ELSIF G_xDoManual THEN
	IF G_xManualActive AND G_xManualEpas AND IFB_RTOPMode.Q THEN
		G_xManualActive := FALSE;
		G_xManualEpas := FALSE;
	ELSIF IFB_RTOPMode.Q THEN
		g_xManualActive := TRUE;
		G_xManualEpas := TRUE;
	END_IF
	G_xJogMachineEpas := FALSE;
	G_xBrakeReleaseEpas := FALSE;
	G_xPrepareEpas:= FALSE;
	G_xAutoEpas := FALSE;

ELSIF g_xDoJogMachine THEN
	IF g_xJogMachineActive AND G_xJogMachineEpas AND IFB_RTOPMode.Q THEN
		g_xJogMachineActive := FALSE;
		G_xJogMachineEpas := FALSE;
	ELSIF IFB_RTOPMode.Q THEN
		g_xJogMachineActive := TRUE;
		G_xJogMachineEpas := TRUE;
	END_IF
	G_xBrakeReleaseEpas := FALSE;
	G_xPrepareEpas:= FALSE;
	G_xAutoEpas := FALSE;
	G_xManualEpas := FALSE;

ELSIF g_xDoBrakeRelease THEN
	IF g_xBrakeReleaseActive AND G_xBrakeReleaseEpas AND IFB_RTOPMode.Q THEN
		g_xBrakeReleaseActive := FALSE;
		G_xBrakeReleaseEpas := FALSE;
	ELSIF IFB_RTOPMode.Q THEN
		g_xBrakeReleaseActive := TRUE;
		G_xBrakeReleaseEpas := TRUE;
	END_IF
	G_xPrepareEpas:= FALSE;
	G_xAutoEpas := FALSE;
	G_xManualEpas := FALSE;
	G_xJogMachineEpas := FALSE;
END_IF

IF g_xDoPrepare OR  g_xDoAuto OR g_xDoManual OR g_xDoJogMachine OR g_xDoBrakeRelease THEN
	g_xPrepareActive := g_xPrepareActive  AND NOT( g_xDoAuto OR g_xDoManual OR g_xDoJogMachine OR g_xDoBrakeRelease);
	g_xAutoActive :=  g_xAutoActive AND NOT( g_xDoPrepare OR g_xDoManual OR g_xDoJogMachine OR g_xDoBrakeRelease);
	g_xManualActive := g_xManualActive AND NOT( g_xDoPrepare OR g_xDoAuto OR g_xDoJogMachine OR g_xDoBrakeRelease);
	g_xJogMachineActive :=  g_xJogMachineActive AND NOT( g_xDoPrepare OR g_xDoAuto OR g_xDoManual OR g_xDoBrakeRelease);
	g_xBrakeReleaseActive:=  g_xBrakeReleaseActive  AND NOT( g_xDoPrepare OR g_xDoAuto OR g_xDoManual OR g_xDoJogMachine);
END_IF
END_ACTION

ACTION SearchCurrentModule:
(* Locate the current module according to the information in audiHierarchy *)
udiCurrentLevel3Size := 0;
pstCurrentFirstLevel3Module := 0;
pstCurrentParent := 0;
dwCurrentAddInterface := 0;
pstCurrent := ADR(SR_MainMachine.stMachineInterface); (* here we have to start at SR_MainMachine.stMachineInterface
instead of our local copy because otherwise it would not be possible to send commands to the MainMachine using the Vis. *)
FOR udiTmp := 2 TO udiCurrentLevel DO
	(* Only navigate to existing modules *)
	IF(pstCurrent^.iq_stExt.udiNumberOfSubModules + pstCurrent^.iq_stExt.udiNumberOfControlModules < audiHierarchy[udiTmp]) THEN
		audiHierarchy[udiTmp] := pstCurrent^.iq_stExt.udiNumberOfSubModules + pstCurrent^.iq_stExt.udiNumberOfControlModules;
	END_IF
	IF(audiHierarchy[udiTmp] <= 0) THEN
		audiHierarchy[udiTmp] := 1;
	END_IF
	IF(pstCurrent^.iq_stExt.udiNumberOfSubModules = 0 AND pstCurrent^.iq_stExt.udiNumberOfControlModules = 0) THEN
		(* Stop, the hierarchy was invalid *)
		udiCurrentLevel := udiTmp - 1;
	ELSE
		(* In case the stSubModules structure of this module is invalid, create an error and stop *)
		IF(pstCurrent^.iq_stExt.dwSubModulesItf = 0) THEN
			stPointerException.sMsg:=						'SR_VisControl: dwSubModuleInterfaces of module was 0';
		END_IF
		IF (pstCurrent^.iq_stExt.pdwSubModulesAddItf = 0 AND pstCurrent^.iq_stExt.dwControlModulesItf = 0) THEN
			stPointerException.sMsg:=						'SR_VisControl: pdwSubModuleAddInterfaces of module was 0';
		END_IF
		(*Set an error if there is no sub module (control module or equipment module)*)
		IF( (pstCurrent^.iq_stExt.dwSubModulesItf = 0 )
			OR (pstCurrent^.iq_stExt.pdwSubModulesAddItf = 0) ) AND pstCurrent^.iq_stExt.dwControlModulesItf = 0 THEN
			(* Error, the structures are not set in the expected way *)
		
			stPointerException.etDiag			:= GD.ET_Diag.UnexpectedProgramBehavior;
			stPointerException.udiDiagExt		:= ET_DiagExt.InvalidPointer;
			stPointerException.sDiagExt			:= FC_EtDiagExtToString(stPointerException.udiDiagExt);
//			stPointerException.sMsg				:= '';
			stPointerException.udiModuleId		:= pstCurrent^.i_udiModuleId;
			stPointerException.sModuleName		:= pstCurrent^.i_sModuleName;
			stPointerException.etSource			:= TPL.ET_ExceptionSource.Vis;
			stPointerException.timDelayTime		:= T#0MS;
			stPointerException.wHmiAttributes	:= 0;
			stPointerException.xAutoQuit		:= FALSE;
			stPointerException.stReaction.axReaction[TPL.ET_Reaction.AsyncStop] := TRUE;

			TPL.FC_SetException(i_xExceptionActive	:= TRUE,
								iq_stException		:= stPointerException,
								iq_stExceptionList	:= G_stExceptionList,
								iq_stLogDataList	:= G_stLogDataList);
								
			xPointerExceptionActive := TRUE;
			RETURN;
		END_IF
		
		pstCurrentParent := pstCurrent;
		(* Only navigate to existing equipment modules *)
		IF pstCurrentParent^.iq_stExt.udiNumberOfSubModules >= audiHierarchy[udiTmp] THEN
			pstCurrent := pstCurrent^.iq_stExt.dwSubModulesItf
				+ UDINT_TO_DWORD((audiHierarchy[udiTmp] - 1) * SIZEOF(vpq_stCurrentModuleStandardInterface));
			IF(udiTmp = 2) THEN
				udiCurrentLevel3Size := pstCurrent^.iq_stExt.udiNumberOfSubModules;
				pstCurrentFirstLevel3Module := pstCurrent^.iq_stExt.dwSubModulesItf;
			END_IF
		END_IF
		(*Initialize pointer for level 2*)
		IF udiTmp = 2 THEN
			pstCurrentLevel2 := pstCurrent;
		END_IF

	END_IF
END_FOR

(*Set pointer to the current module interface*)
IF pstCurrentParent = 0  THEN
	pstCurrentControlModuleStandardInterface 	:= pstCurrent^.iq_stExt.dwControlModulesItf;
	udiCurrentNumberOfControlModules 			:= pstCurrent^.iq_stExt.udiNumberOfControlModules;
ELSE
	pstCurrentControlModuleStandardInterface 	:= pstCurrentParent^.iq_stExt.dwControlModulesItf;
	udiCurrentNumberOfControlModules 			:= pstCurrentParent^.iq_stExt.udiNumberOfControlModules;
END_IF
IF pstCurrentLevel2 <> 0 THEN
	udiNumberOfControlModulesLevel2:= pstCurrentLevel2^.iq_stExt.udiNumberOfControlModules;
ELSE
	udiNumberOfControlModulesLevel2:= 0;
END_IF
END_ACTION

ACTION SetCurrentModule:
(*
	handles all requests coming from the special vis controllers

	sets the current module by modifying aiHierachy
	also sets the jog target

inputs:
	diSetAsCurrentModule - if <> 0 contains the module ID of the module to set as current module

in_out:
	audiHierarchy	
	udiCurrentLevel

flags:
	

*)
IF(udiSetAsCurrentModule > 0) THEN
	udiTmp2 := 1;
	WHILE(udiSetAsCurrentModule > udiTmp2 * 100) DO
		udiTmp2 := udiTmp2 * 100;
	END_WHILE

	udiCurrentLevel := 0;
	WHILE(udiTmp2 > 0) DO
		udiCurrentLevel := udiCurrentLevel + 1;
		audiHierarchy[udiCurrentLevel] := udiSetAsCurrentModule / udiTmp2;
		udiSetAsCurrentModule := udiSetAsCurrentModule MOD udiTmp2;
		udiTmp2 := udiTmp2 / 100;
	END_WHILE

	IF(udiCurrentLevel < 1) THEN
		udiCurrentLevel := 1;
	END_IF

	udiSetAsCurrentModule := 0;
	xUpdateData := TRUE;
END_IF

IF(udiSetAsJogTarget <> 0) THEN
	G_udiManualModuleSelect		:= udiSetAsJogTarget;
//	G_udiManualElementSelect	:= udiSetAsJogTargetNum;
	udiSetAsJogTarget := 0;
//	udiSetAsJogTargetNum := 0;
END_IF
END_ACTION

END_PROGRAM

// LMC_PacDrive/Application/FB_ExampleLeafModuleVisController
FUNCTION_BLOCK FB_ExampleLeafModuleVisController

VAR_INPUT
	i_xEnable								: BOOL;
	i_pstMachineStandardItf					: POINTER TO TPL.ST_StandardModuleInterface;
	i_pstCurrentStandardItf					: POINTER TO TPL.ST_StandardModuleInterface;
	i_dwCurrentAddItf						: DWORD;
	i_xUpdateData							: BOOL; (* Signals the selection of another module *)
	i_udiCurrentJogTarget					: UDINT;
END_VAR

VAR_IN_OUT
	iq_stExceptionList				: TPL.ST_ExceptionList;
	iq_stLogDataList	   			: TPL.ST_LogDataList;
END_VAR

VAR_OUTPUT
	q_xActive								: BOOL;
	q_xReady								: BOOL;
	q_etDiag								: GD.ET_Diag := GD.ET_Diag.Ok;
	q_etDiagExt								: ET_DiagExtExampleLeafModule := ET_DiagExtExampleLeafModule.Disabled;
	q_sMsg									: STRING[80] := '';
	q_udiSetAsCurrentModule					: UDINT; (* A moduleID, if <> 0, it is set as the current module *)
	q_udiSetAsJogTarget						: UDINT;
END_VAR

VAR
	xCurrentIsOfMyType						: BOOL;
	pstCurrentExampleLeafModuleInterface	: POINTER TO ST_ExampleLeafModuleInterface;
	stCurrentExampleLeafModuleInterface		: ST_ExampleLeafModuleInterface;
	iPaneSelect								: INT := 1; (* Variable for selecting the active pane *)

	(* Variables to detect user changes in the vis *)
	xInitUserInputs							: BOOL;

	(* list of all example leaf modules in the machine *)
	audiExampleLeafModuleId					: ARRAY[1..c_udiMaxExampleLeafModules] OF UDINT; (* if <> 0, module exists *)
	asExampleLeafModuleName					: ARRAY[1..c_udiMaxExampleLeafModules] OF STRING[80]; (* if <> 0, module exists *)
	udiCountExampleLeafModules				: UDINT;
	udiSetAsCurrentModule					: UDINT;

	(* temporary variable, not to be used after init *)
	apExampleLeafModuleInterface			: ARRAY[1..c_udiMaxExampleLeafModules] OF POINTER TO TPL.ST_StandardModuleInterface;
	udiTmp									: UDINT;
	xEnableFlag								: BOOL;

	(* Variables to detect user changes in the vis *)
	lrPosMax								: LREAL;
END_VAR

VAR CONSTANT
	c_udiMaxExampleLeafModules : UDINT := 10;
END_VAR

q_udiSetAsCurrentModule 	:= 0;
q_udiSetAsJogTarget			:= 0;

(*********************************************************************)

IF i_xEnable AND NOT xEnableFlag THEN
	xEnableFlag := TRUE;
	
	q_xActive	:= TRUE;	
	
	q_etDiag	:= GD.ET_Diag.Ok;
	q_etDiagExt := ET_DiagExtExampleLeafModule.Initializing;
	q_sMsg		:= '';
	
	
		
	udiCountExampleLeafModules := TPL.FC_GetAllModulesOfType(	i_pstMachineStandardItf	:= i_pstMachineStandardItf,
																i_dwWantedType			:= ET_ModuleType.ExampleLeafModule,  
																i_pdwResultSet			:= ADR(apExampleLeafModuleInterface), 
																i_udiResultSetSize		:= c_udiMaxExampleLeafModules);
	FOR udiTmp := 1 TO udiCountExampleLeafModules DO
		(* module version check *)
		IF(apExampleLeafModuleInterface[udiTmp]^.q_udiModuleVersion = 1) THEN
			audiExampleLeafModuleId[udiTmp] := apExampleLeafModuleInterface[udiTmp]^.i_udiModuleId;
			asExampleLeafModuleName[udiTmp] := apExampleLeafModuleInterface[udiTmp]^.i_sModuleName;
		END_IF
	END_FOR
	
	q_xReady	:= TRUE;
	
	q_etDiag	:= GD.ET_Diag.Ok;
	q_etDiagExt	:= ET_DiagExtExampleLeafModule.Working;
	q_sMsg		:= '';
	
ELSIF NOT i_xEnable AND xEnableFlag THEN
	xEnableFlag := FALSE;
	
	q_xActive				:= FALSE;	
	q_xReady				:= FALSE;
	q_etDiag				:= GD.ET_Diag.Ok;
	q_etDiagExt				:= ET_DiagExtExampleLeafModule.Disabled;
	q_sMsg					:= '';
	q_udiSetAsCurrentModule	:= 0;		
	q_udiSetAsJogTarget		:= 0;		
END_IF

IF i_xEnable THEN
	q_udiSetAsCurrentModule := udiSetAsCurrentModule;
	udiSetAsCurrentModule := 0;
END_IF


(*********************************************************************)


IF i_xEnable THEN
	IF i_pstCurrentStandardItf = 0 THEN
		q_xReady := FALSE;
		q_etDiag := GD.ET_Diag.InputParameterInvalid;
		q_etDiagExt := ET_DiagExtExampleLeafModule.CurrentStandardItfInvalidPointer;
		q_sMsg := '';
	ELSIF i_dwCurrentAddItf = 0 THEN
		q_xReady := FALSE;
		q_etDiag := GD.ET_Diag.InputParameterInvalid;
		q_etDiagExt := ET_DiagExtExampleLeafModule.CurrentAddItfInvalidPointer;
		q_sMsg := '';
	ELSE
		q_xReady	:= TRUE;
	
		q_etDiag	:= GD.ET_Diag.Ok;
		q_etDiagExt	:= ET_DiagExtExampleLeafModule.Working;
		q_sMsg		:= '';
		
		IF (i_pstCurrentStandardItf^.q_dwModuleType = UDINT_TO_DWORD(ET_ModuleType.ExampleLeafModule)) THEN
			(* Module version check *)
			IF(i_pstCurrentStandardItf^.q_udiModuleVersion = 1) THEN
				pstCurrentExampleLeafModuleInterface := i_dwCurrentAddItf;
				xCurrentIsOfMyType := TRUE;
			END_IF
		ELSE
			pstCurrentExampleLeafModuleInterface := 0;
			xCurrentIsOfMyType := FALSE;
		END_IF	
	
		IF(xCurrentIsOfMyType) THEN
			(* Execute changes requested by user first *)
			IF(NOT xInitUserInputs) THEN
				xInitUserInputs := TRUE;
				(* Ignore values of variables now *)
			ELSE
				(* Detect user changes *)
				IF stCurrentExampleLeafModuleInterface.i_lrPosMax <> lrPosMax THEN
					pstCurrentExampleLeafModuleInterface^.i_lrPosMax := stCurrentExampleLeafModuleInterface.i_lrPosMax;
				END_IF
	
				(* ... *)
			END_IF
			stCurrentExampleLeafModuleInterface := pstCurrentExampleLeafModuleInterface^;
	
		ELSE
			;
			(* Reset other flags *)
		END_IF
	END_IF
ELSE
	xCurrentIsOfMyType := FALSE;
END_IF

END_FUNCTION_BLOCK

// GetBooleanProperty
// This function has been automatically generated from the project information.
{attribute 'signature_flag' := '1073741824'}
{attribute 'register_in_runtime'}
FUNCTION GetBooleanProperty : BOOL
VAR_INPUT
	stKey: WSTRING;
END_VAR

GetBooleanProperty := FALSE;

END_FUNCTION

// GetTextProperty2
// This function has been automatically generated from the project information.
{attribute 'signature_flag' := '1073741824'}
{attribute 'register_in_runtime'}
FUNCTION GetTextProperty2 : POINTER TO WSTRING
VAR_INPUT
	stKey: WSTRING;
END_VAR

IF stKey = "Author" THEN
	GetTextProperty2 := ADR("SESA110233");
ELSIF stKey = "Company" THEN
	GetTextProperty2 := ADR("");
ELSIF stKey = "DefaultNamespace" THEN
	GetTextProperty2 := ADR("CrankModuleExample");
ELSIF stKey = "Description" THEN
	GetTextProperty2 := ADR("");
ELSIF stKey = "Project" THEN
	GetTextProperty2 := ADR("Template_GitHub_ESME22");
ELSIF stKey = "Title" THEN
	GetTextProperty2 := ADR("Template_GitHub_ESME22");
ELSE
	GetTextProperty2 := ADR("");
END_IF

END_FUNCTION

// GetTextProperty
// This function has been automatically generated from the project information.
{attribute 'signature_flag' := '1073741824'}
{attribute 'register_in_runtime'}
FUNCTION GetTextProperty : WSTRING
VAR_INPUT
	stKey: WSTRING;
END_VAR

IF stKey = "Author" THEN
	GetTextProperty := "SESA110233";
ELSIF stKey = "Company" THEN
	GetTextProperty := "";
ELSIF stKey = "DefaultNamespace" THEN
	GetTextProperty := "CrankModuleExample";
ELSIF stKey = "Description" THEN
	GetTextProperty := "";
ELSIF stKey = "Project" THEN
	GetTextProperty := "Template_GitHub_ESME22";
ELSIF stKey = "Title" THEN
	GetTextProperty := "Template_GitHub_ESME22";
ELSE
	GetTextProperty := "";
END_IF

END_FUNCTION

// GetTitle
// This function has been automatically generated from the project information.
{attribute 'signature_flag' := '1073741824'}
{attribute 'register_in_runtime'}
FUNCTION GetTitle : WSTRING
VAR_INPUT
	
END_VAR

GetTitle := "Template_GitHub_ESME22";

END_FUNCTION

// LMC_PacDrive/Application/CheckBounds
// Implicitly generated code : DO NOT EDIT
FUNCTION CheckBounds : DINT
VAR_INPUT
	index, lower, upper: DINT;
END_VAR

IF  index < lower THEN
	CheckBounds := lower;
	FC_DiagMsgWrite(4, CONCAT('CB min>', CONCAT('idx=', DINT_TO_STRING(index))));
	FC_SysUserCallStack(0);
ELSIF  index > upper THEN
	CheckBounds := upper;
	FC_DiagMsgWrite(4, CONCAT('CB max<', CONCAT('idx=', DINT_TO_STRING(index))));
	FC_SysUserCallStack(0);
ELSE  
	CheckBounds := index;
END_IF

END_FUNCTION

// LMC_PacDrive/Application/CheckDivDInt
// Implicitly generated code : DO NOT EDIT
FUNCTION CheckDivDInt : DINT
VAR_INPUT
	divisor: DINT;
END_VAR

IF divisor = 0 THEN
	CheckDivDInt:=1;
	FC_DiagMsgWrite(4, 'CDDI Div by 0');
	FC_SysUserCallStack(0);
ELSE
	CheckDivDInt:=divisor;
END_IF

END_FUNCTION

// LMC_PacDrive/Application/CheckDivLInt
// Implicitly generated code : DO NOT EDIT
FUNCTION CheckDivLInt : LINT
VAR_INPUT
	divisor: LINT;
END_VAR

IF divisor = 0 THEN
	CheckDivLInt:=1;
	FC_DiagMsgWrite(4, 'CDLI Div by 0');
	FC_SysUserCallStack(0);
ELSE
	CheckDivLInt:=divisor;
END_IF

END_FUNCTION

// LMC_PacDrive/Application/CheckDivLReal
// Implicitly generated code : DO NOT EDIT
FUNCTION CheckDivLReal : LREAL
VAR_INPUT
	divisor: LREAL;
END_VAR

IF divisor = 0 THEN
	CheckDivLReal:=1;
	FC_DiagMsgWrite(4, 'CDLR Div by 0');
	FC_SysUserCallStack(0);
ELSE
	CheckDivLReal:=divisor;
END_IF

END_FUNCTION

// LMC_PacDrive/Application/CheckDivReal
// Implicitly generated code : DO NOT EDIT
FUNCTION CheckDivReal : REAL
VAR_INPUT
	divisor: REAL;
END_VAR

IF divisor = 0 THEN
	CheckDivReal:=1;
	FC_DiagMsgWrite(4, 'CDR Div by 0');
	FC_SysUserCallStack(0);
ELSE
	CheckDivReal:=divisor;
END_IF

END_FUNCTION

// LMC_PacDrive/Application/CheckLRangeSigned
// Implicitly generated code : DO NOT EDIT
FUNCTION CheckLRangeSigned : LINT
VAR_INPUT
	value, lower, upper: LINT;
END_VAR

IF (value < lower) THEN
	CheckLRangeSigned := lower;
	FC_DiagMsgWrite(4, CONCAT('CLRS min>', CONCAT('idx=', LINT_TO_STRING(value))));
	FC_SysUserCallStack(0);
ELSIF(value > upper) THEN
	CheckLRangeSigned := upper;
	FC_DiagMsgWrite(4, CONCAT('CLRS max<', CONCAT('idx=', LINT_TO_STRING(value))));
	FC_SysUserCallStack(0);
ELSE
	CheckLRangeSigned := value;
END_IF

END_FUNCTION

// LMC_PacDrive/Application/CheckLRangeUnsigned
// Implicitly generated code : DO NOT EDIT
FUNCTION CheckLRangeUnsigned : ULINT
VAR_INPUT
	value, lower, upper: ULINT;
END_VAR

IF (value < lower) THEN
	CheckLRangeUnsigned := lower;
	FC_DiagMsgWrite(4, CONCAT('CLRU min>', CONCAT('idx=', ULINT_TO_STRING(value))));
	FC_SysUserCallStack(0);
ELSIF(value > upper) THEN
	CheckLRangeUnsigned := upper;
	FC_DiagMsgWrite(4, CONCAT('CLRU max<', CONCAT('idx=', ULINT_TO_STRING(value))));
	FC_SysUserCallStack(0);
ELSE
	CheckLRangeUnsigned := value;
END_IF

END_FUNCTION

// LMC_PacDrive/Application/CheckPointer
// Implicitly generated code : DO NOT EDIT
FUNCTION CheckPointer : POINTER TO BYTE
VAR_INPUT
	ptToTest: POINTER TO BYTE; // Destination address of the pointer
	iSize: DINT;            // Size of the type the pointer points to. (e.g: 20 for POINTER TO ARRAY [0..9] OF INT)
	iGran: DINT;		// Granularity of the pointer access. This is the size of the biggest non-structured data type in the type the pointer points to. (e.g: 2 for POINTER TO ARRAY [0..9] OF INT)
	bWrite: BOOL;		// Indicates read or write Access. TRUE = write access.
END_VAR

CheckPointer := ptToTest;
IF ptToTest = 0 THEN
	FC_DiagMsgWrite(4, 'CP = 0');
	FC_SysUserCallStack(0);
ELSE
	CheckPointer := ptToTest;
END_IF

END_FUNCTION

// LMC_PacDrive/Application/CheckRangeSigned
// Implicitly generated code : DO NOT EDIT
FUNCTION CheckRangeSigned : DINT
VAR_INPUT
	value, lower, upper: DINT;
END_VAR

IF (value < lower) THEN
	CheckRangeSigned := lower;
	FC_DiagMsgWrite(4, CONCAT('CRS min>', CONCAT('idx=', DINT_TO_STRING(value))));
	FC_SysUserCallStack(0);
ELSIF(value > upper) THEN
	CheckRangeSigned := upper;
	FC_DiagMsgWrite(4, CONCAT('CRS max<', CONCAT('idx=', DINT_TO_STRING(value))));
	FC_SysUserCallStack(0);
ELSE
	CheckRangeSigned := value;
END_IF

END_FUNCTION

// LMC_PacDrive/Application/CheckRangeUnsigned
// Implicitly generated code : DO NOT EDIT
FUNCTION CheckRangeUnsigned : UDINT
VAR_INPUT
	value, lower, upper: UDINT;
END_VAR

IF (value < lower) THEN
	CheckRangeUnsigned := lower;
	FC_DiagMsgWrite(4, CONCAT('CRU min>', CONCAT('idx=', UDINT_TO_STRING(value))));
	FC_SysUserCallStack(0);
ELSIF(value > upper) THEN
	CheckRangeUnsigned := upper;
	FC_DiagMsgWrite(4, CONCAT('CRU max<', CONCAT('idx=', UDINT_TO_STRING(value))));
	FC_SysUserCallStack(0);
ELSE
	CheckRangeUnsigned := value;
END_IF

END_FUNCTION

// LMC_PacDrive/Application/CrankModuleExample/Examples/ExampleModulesExtItf/FB_ExampleLeafModuleExtItf
FUNCTION_BLOCK FB_ExampleLeafModuleExtItf

VAR_INPUT
(* Part of TPL.ST_StandardModuleInterface.i_... *)
	i_xEnable						: BOOL;			
END_VAR

VAR_IN_OUT
(* Part of TPL.ST_StandardModuleInterface.iq_... *)
	iq_diCmd						: DINT;

(* TPL.ST_StandardModuleInterface *)	
	iq_stStandardModuleItf			: TPL.ST_StandardModuleInterface;
	
(* ExceptionHandling and Logging *)	
	iq_stExceptionList				: TPL.ST_ExceptionList;
	iq_stLogDataList				: TPL.ST_LogDataList;
	
(* ST_ExampleLeafModuleInterface *)
	iq_stExampleLeafModuleItf		: ST_ExampleLeafModuleInterface;
END_VAR

VAR_OUTPUT
(* TPL.ST_StandardModuleInterface.q_... *)
	q_xActive						: BOOL;
	q_xReady						: BOOL;
	q_etDiag						: GD.ET_Diag; 
	q_etDiagExt						: ET_DiagExtExampleLeafModule;
	q_sMsg							: STRING[80];
	q_xCmdActive					: BOOL;
	q_diCmdActive					: DINT;
	q_xCmdDone						: BOOL;	
END_VAR

VAR
	fbExampleLeafModule : FB_ExampleLeafModule;
END_VAR

(* System generated code, could be modified for your application *)

iq_stStandardModuleItf.i_xEnable	:= i_xEnable;
iq_stStandardModuleItf.iq_diCmd		:= iq_diCmd;

(* Module call *)
fbExampleLeafModule(iq_stStandardModuleItf		:= iq_stStandardModuleItf, 
					iq_stExceptionList			:= iq_stExceptionList, 
					iq_stLogDataList			:= iq_stLogDataList, 
					iq_stExampleLeafModuleItf	:= iq_stExampleLeafModuleItf);
					
iq_diCmd	:= iq_stStandardModuleItf.iq_diCmd;

q_xActive		:= iq_stStandardModuleItf.q_xActive;
q_xReady		:= iq_stStandardModuleItf.q_xReady;
q_etDiag		:= iq_stStandardModuleItf.q_etDiag; 
q_etDiagExt		:= iq_stStandardModuleItf.q_udiDiagExt;
q_sMsg			:= iq_stStandardModuleItf.q_sMsg;
q_xCmdActive	:= iq_stStandardModuleItf.q_xCmdActive;
q_diCmdActive	:= iq_stStandardModuleItf.q_diCmdActive;
q_xCmdDone		:= iq_stStandardModuleItf.q_xCmdDone;	

(* End of system generated code, could be modified for your application *)

END_FUNCTION_BLOCK

// LMC_PacDrive/Application/CrankModuleExample/Examples/ExampleModulesExtItf/FB_ExampleNodeFbModuleExtItf
FUNCTION_BLOCK FB_ExampleNodeFbModuleExtItf

VAR_INPUT
(* Part of TPL.ST_StandardModuleInterface.i_... *)
	i_xEnable						: BOOL;
	
(* Master of ExampleNodeFbModule *)
	i_ifMaster						: SystemConfigurationItf.IF_Master;
END_VAR

VAR_IN_OUT
(* Part of TPL.ST_StandardModuleInterface.iq_... *)
	iq_diCmd						: DINT;
	iq_diStartStep					: DINT;

(* TPL.ST_StandardModuleInterface *)	
	iq_stStandardModuleItf			: TPL.ST_StandardModuleInterface;
	
(* TPL.ST_StandardMotionInterface *)		
	iq_stStandardMotionItf			: TPL.ST_StandardMotionInterface;
	
(* Additional interface *)
	iq_stAdditionalItf				: ST_ExampleNodeAsFbInterface;
	
(* ExceptionHandling and Logging *)	
	iq_stExceptionList				: TPL.ST_ExceptionList;
	iq_stLogDataList				: TPL.ST_LogDataList;
END_VAR

VAR_OUTPUT
(* Part of TPL.ST_StandardModuleInterface.q_... *)
	q_xActive						: BOOL;
	q_xReady						: BOOL;
	q_etDiag						: GD.ET_Diag; 
	q_etDiagExt						: ET_DiagExt;
	q_sMsg							: STRING[80];	
	q_xCmdActive					: BOOL;
	q_diCmdActive					: DINT;
	q_xCmdDone						: BOOL;
	q_udiActiveSubModule			: UDINT;
	q_udiSubModuleInException		: UDINT;
END_VAR

VAR
	fbExampleNodeFbModule : FB_ExampleNodeFbModule;
END_VAR

(* System generated code, could be modified for your application *)

iq_stStandardModuleItf.i_xEnable		:= i_xEnable;
iq_stStandardModuleItf.iq_diCmd			:= iq_diCmd;
iq_stStandardModuleItf.iq_diStartStep	:= iq_diStartStep;

(* Module call *)
fbExampleNodeFbModule(	i_ifMaster				:= i_ifMaster, 
						iq_stStandardModuleItf	:= iq_stStandardModuleItf, 
						iq_stStandardMotionItf	:= iq_stStandardMotionItf, 
						iq_stAdditionalItf		:= iq_stAdditionalItf, 
						iq_stExceptionList		:= iq_stExceptionList, 
						iq_stLogDataList		:= iq_stLogDataList);
						
iq_diCmd		:= iq_stStandardModuleItf.iq_diCmd;
iq_diStartStep	:= iq_stStandardModuleItf.iq_diStartStep;

q_xActive					:= iq_stStandardModuleItf.q_xActive;
q_xReady					:= iq_stStandardModuleItf.q_xReady;
q_etDiag					:= iq_stStandardModuleItf.q_etDiag; 
q_etDiagExt					:= iq_stStandardModuleItf.q_udiDiagExt;
q_sMsg						:= iq_stStandardModuleItf.q_sMsg;	
q_xCmdActive				:= iq_stStandardModuleItf.q_xCmdActive;
q_diCmdActive				:= iq_stStandardModuleItf.q_diCmdActive;
q_xCmdDone					:= iq_stStandardModuleItf.q_xCmdDone;
q_udiActiveSubModule		:= iq_stStandardModuleItf.q_udiActiveSubModule;
q_udiSubModuleInException	:= iq_stStandardModuleItf.q_udiSubModuleInException;

(* End of system generated code, could be modified for your application *)

END_FUNCTION_BLOCK

// LMC_PacDrive/Application/CrankModuleExample/Examples/ExampleNodeAsFB/FB_ExampleNodeFbModule
FUNCTION_BLOCK FB_ExampleNodeFbModule

VAR CONSTANT
(* Standard related constants *)
	c_udiNumberOfGroups				: UDINT := 3;			(* Maximum number of groups *)
	c_udiNumberOfGroupMembers		: UDINT := 10;			(* Maximum number of members per group *)

	c_udiNumberOfCmdTables			: UDINT := 8;			(* Must be the exact number of used CMDTables! *)
	c_udiNumberOfCmdSteps			: UDINT := 16;			(* Make sure that the number of steps per command that each table
															   contains does not exceed the c_diNumberOfCmdSteps variable. *)

(*Definition group of modules *)
	c_udiSlaveGroup1				: UDINT := 2001;		(* Name of module group  1 *)
	c_udiSlaveGroup2				: UDINT := 2002;		(* Name of module group  2 *)

(* System generated code, could be modified for your application *)
	c_udiNumberOfSubModules			: UDINT := 2;				(* Number of axis modules *)
	c_udiSlave1						: UDINT := 1;
	c_udiSlave2						: UDINT := 2;
(* End of system generated code, could be modified for your application *)
END_VAR

VAR	(* User specific variables *)
	stSlave1Interface				: AXM.ST_ModuleInterface;
	fbSlave1Module					: AXM.FB_AxisModule;
	
	stSlave2Interface				: AXM.ST_ModuleInterface;
	fbSlave2Module					: AXM.FB_AxisModule;
	
	fbAxixModuleController			: AXM.FB_AxisModuleController;
END_VAR

VAR_INPUT
(* Master of ExampleNodeFbModule *)
	i_ifMaster						: SystemConfigurationItf.IF_Master;
END_VAR

VAR_IN_OUT
(* TPL.ST_StandardModuleInterface *)	
	iq_stStandardModuleItf			: TPL.ST_StandardModuleInterface;
	
(* TPL.ST_StandardMotionInterface *)		
	iq_stStandardMotionItf			: TPL.ST_StandardMotionInterface;
	
(* Additional interface *)
	iq_stAdditionalItf				: ST_ExampleNodeAsFbInterface;
	
(* ExceptionHandling and Logging *)	
	iq_stExceptionList				: TPL.ST_ExceptionList;
	iq_stLogDataList				: TPL.ST_LogDataList;
END_VAR

VAR
	xInitSuccessful : BOOL := TRUE;
		
(* Standard related variables *)
	astSubModuleInterface			: ARRAY[1..c_udiNumberOfSubModules] OF TPL.ST_StandardModuleInterface;		(* Interface to modules *)
	aaudiSubModuleGroups			: ARRAY[1..c_udiNumberOfGroups,1..c_udiNumberOfGroupMembers] OF UDINT;
	adwSubModuleAddInterfaces		: ARRAY[1..c_udiNumberOfSubModules] OF DWORD;

(* Modules related variables *)
	fbModuleController				: TPL.FB_ModuleController;
	etDiagModuleController			: GD.ET_Diag;
	etDiagExtModuleController		: TPL.ET_DiagExt;
	sMsgModuleController			: STRING[80];
	xWaitForStartStep				: BOOL;

	astListOfCmdTables				: ARRAY [1..c_udiNumberOfCmdTables] OF TPL.ST_CmdTable;
	udiTableIndex					: UDINT;
	udiStepIndex					: UDINT;
	diStep							: DINT;

	astPrepareTable					: ARRAY [1..c_udiNumberOfCmdSteps] OF TPL.ST_Cmd;		(* Relating  Cmd table *)
	astAutoTable					: ARRAY [1..c_udiNumberOfCmdSteps] OF TPL.ST_Cmd;		(* Relating  Cmd table *)
	astManualTable					: ARRAY [1..c_udiNumberOfCmdSteps] OF TPL.ST_Cmd;		(* Relating  Cmd table *)
	astHoldTable					: ARRAY [1..c_udiNumberOfCmdSteps] OF TPL.ST_Cmd;		(* Relating  Cmd table *)
	astStartTable					: ARRAY [1..c_udiNumberOfCmdSteps] OF TPL.ST_Cmd;		(* Relating  Cmd table *)
	astStopTable					: ARRAY [1..c_udiNumberOfCmdSteps] OF TPL.ST_Cmd;		(* Relating  Cmd table *)
	astBrakeReleaseTable			: ARRAY [1..c_udiNumberOfCmdSteps] OF TPL.ST_Cmd;		(* Relating  Cmd table *)
	astAbortTable					: ARRAY [1..c_udiNumberOfCmdSteps] OF TPL.ST_Cmd;		(* Relating  Cmd table *)

(* ExceptionHandling related variables *)
	fbExceptionHandler				: TPL.FB_ExceptionHandler;

	aetReactionTranslationMode		: ARRAY[1..c_udiNumberOfSubModules] OF TPL.ET_ReactionTranslationMode;
	aastReactionTranslationTable	: ARRAY[1..c_udiNumberOfSubModules,1..TPL.Gc_udiMaxNumberOfReactions] OF TPL.ST_Reaction;
	astReactionTranslationJobs		: ARRAY[1..c_udiNumberOfSubModules] OF TPL.ST_ReactionTranslationJobs;

(* Exception declaration *)
	stUserException1				: TPL.ST_Exception;
	stUserException2				: TPL.ST_Exception;
	xModuleUserException1			: BOOL;
	xModuleUserException2			: BOOL;
	
	stUpdateStructsException		: TPL.ST_Exception;
	xUpdateStructsException			: BOOL;
	
	stInitReactionsException		: TPL.ST_Exception;
	xInitReactionsException			: BOOL;
	
	stInitSubModulesException		: TPL.ST_Exception;
	xInitSubModulesException		: BOOL;
	
	stIsDriveVirtualException		: TPL.ST_Exception;
	xIsDriveVirtualException		: BOOL;

(* Logging related variables*)
	fbLogger						: TPL.FB_Logger;

(* OnlineChange related variables *)
	fbDetectOnlineChange			: TPL.FB_DetectOnlineChange;
	xDetectOnlineChangeActive		: BOOL; 
	xDetectOnlineChangeReady		: BOOL; 
	etDetectOnlineChangeDiag		: GD.ET_Diag;
	etDetectOnlineChangeDiagExt		: TPL.ET_DiagExt; 
	sDetectOnlineChangeMsg			: STRING[80];
	
(* Init related variables *)	
	stLogicalAddressMaster			: SystemConfigurationItf.ST_LogicalAddress;
	lrShaftRefDelay					: LREAL;
	diResult						: DINT;	
	
	xDriveIsVirtual					: BOOL;	
	
(* POU-Feedback related variables*)	
	etDiag			: GD.ET_Diag;
	etDiagExtTPL	: TPL.ET_DiagExt;
	etDiagExtAXM	: AXM.ET_DiagExt;
	sMsgBuffer		: STRING[80];
END_VAR

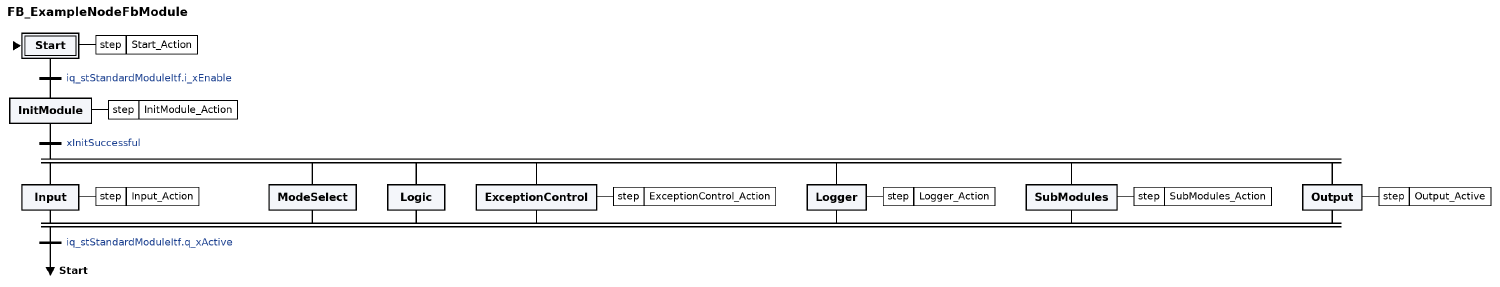
INITIAL_STEP Start:
    Start_Action(N);  // step action
END_STEP
TRANSITION FROM Start TO InitModule
    := iq_stStandardModuleItf.i_xEnable;
END_TRANSITION
STEP InitModule:
    InitModule_Action(N);  // step action
END_STEP
TRANSITION FROM InitModule TO (Input, ModeSelect, Logic, ExceptionControl, Logger, SubModules, Output)
    := xInitSuccessful;
END_TRANSITION
STEP Input:
    Input_Action(N);  // step action
END_STEP
STEP ModeSelect:
END_STEP
STEP Logic:
END_STEP
STEP ExceptionControl:
    ExceptionControl_Action(N);  // step action
END_STEP
STEP Logger:
    Logger_Action(N);  // step action
END_STEP
STEP SubModules:
    SubModules_Action(N);  // step action
END_STEP
STEP Output:
    Output_Active(N);  // step action
END_STEP
TRANSITION FROM (Input, ModeSelect, Logic, ExceptionControl, Logger, SubModules, Output) TO Start
    := iq_stStandardModuleItf.q_xActive;
END_TRANSITION

ACTION ExceptionControl_Action:
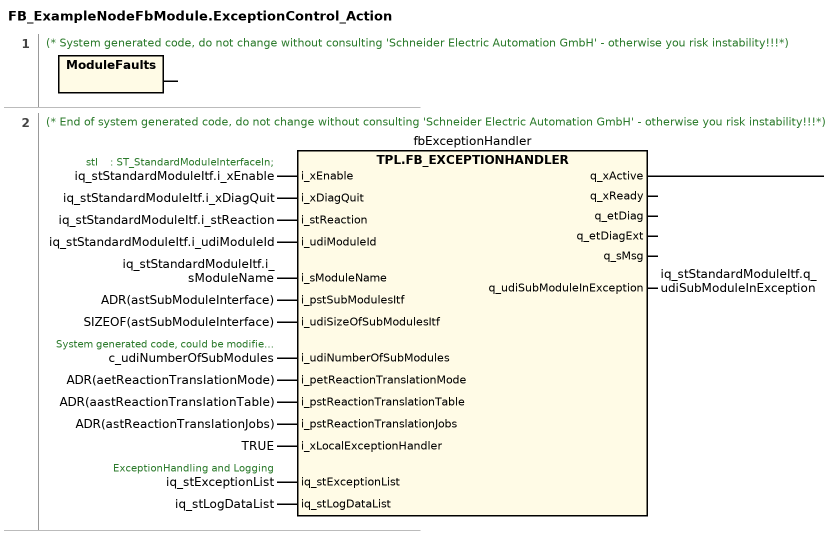
// NETWORK 1
// 					(* System generated code, do not change without consulting 'Schneider Electric Automation GmbH' - otherwise you risk instability!!!*)
//
//
ModuleFaults();

// NETWORK 2
// (* End of system generated code, do not change without consulting 'Schneider Electric Automation GmbH' - otherwise you risk instability!!!*)
//   fbExceptionHandler: ExceptionHandling related variables
//   iq_stStandardModuleItf.i_xEnable: stI : ST_StandardModuleInterfaceIn;
//   c_udiNumberOfSubModules: System generated code, could be modified for your application
//   iq_stExceptionList: ExceptionHandling and Logging
fbExceptionHandler(
    i_xEnable := iq_stStandardModuleItf.i_xEnable,
    i_xDiagQuit := iq_stStandardModuleItf.i_xDiagQuit,
    i_stReaction := iq_stStandardModuleItf.i_stReaction,
    i_udiModuleId := iq_stStandardModuleItf.i_udiModuleId,
    i_sModuleName := iq_stStandardModuleItf.i_sModuleName,
    i_pstSubModulesItf := ADR(astSubModuleInterface),
    i_udiSizeOfSubModulesItf := SIZEOF(astSubModuleInterface),
    i_udiNumberOfSubModules := c_udiNumberOfSubModules,
    i_petReactionTranslationMode := ADR(aetReactionTranslationMode),
    i_pstReactionTranslationTable := ADR(aastReactionTranslationTable),
    i_pstReactionTranslationJobs := ADR(astReactionTranslationJobs),
    i_xLocalExceptionHandler := TRUE,
    iq_stExceptionList := iq_stExceptionList,
    iq_stLogDataList := iq_stLogDataList,
    q_udiSubModuleInException => iq_stStandardModuleItf.q_udiSubModuleInException); // TPL.FB_EXCEPTIONHANDLER
END_ACTION

ACTION Init_CmdTables:
(* System generated code, could be modified for your application *)

(*********************************************************************************************************************)
(*** Prepare  ***)

TPL.FC_FirstStep(udiStepIndex, diStep);
astPrepareTable[udiStepIndex].sTitle					:= 'DriveEnable On Slave1';
astPrepareTable[udiStepIndex].udiModuleName				:= c_udiSlave1;
astPrepareTable[udiStepIndex].diStep					:= diStep;
astPrepareTable[udiStepIndex].diCmd						:= AXM.ET_Cmd.DriveEnableOn;
astPrepareTable[udiStepIndex].timTimeOut				:= T#0MS;
astPrepareTable[udiStepIndex].xEndCmd					:= FALSE;

TPL.FC_NextStep(udiStepIndex, diStep);
astPrepareTable[udiStepIndex].sTitle					:= 'Homing Mode Slave1';
astPrepareTable[udiStepIndex].udiModuleName				:= c_udiSlave1;
astPrepareTable[udiStepIndex].diStep					:= diStep;
astPrepareTable[udiStepIndex].diCmd						:= AXM.ET_Cmd.Homing;
astPrepareTable[udiStepIndex].timTimeOut				:= T#0MS;
astPrepareTable[udiStepIndex].xEndCmd					:= FALSE;

TPL.FC_NextStep(udiStepIndex, diStep);
astPrepareTable[udiStepIndex].sTitle					:= 'Homing Start Slave1';
astPrepareTable[udiStepIndex].udiModuleName				:= c_udiSlave1;
astPrepareTable[udiStepIndex].diStep					:= diStep;
astPrepareTable[udiStepIndex].diCmd						:= AXM.ET_Cmd.Start;
astPrepareTable[udiStepIndex].timTimeOut				:= T#0MS;
astPrepareTable[udiStepIndex].xEndCmd					:= FALSE;

TPL.FC_LastStep(udiStepIndex, diStep);
astPrepareTable[udiStepIndex].sTitle					:= 'End';
astPrepareTable[udiStepIndex].udiModuleName				:= 0;
astPrepareTable[udiStepIndex].diStep					:= diStep;
astPrepareTable[udiStepIndex].diCmd						:= 0;
astPrepareTable[udiStepIndex].timTimeOut				:= T#0MS;
astPrepareTable[udiStepIndex].xEndCmd					:= TRUE;

TPL.FC_FirstCmdTable(iq_udiTableIndex := udiTableIndex);
astListofCMDTables[udiTableIndex].sTitle				:= 'Prepare';
astListofCMDTables[udiTableIndex].diCmd					:= ET_Cmd.Prepare;
astListofCMDTables[udiTableIndex].udiNumberOfCmdSteps	:= udiStepIndex;

(*********************************************************************************************************************)
(*** Auto  ***)

TPL.FC_FirstStep(udiStepIndex, diStep);
astAutoTable[udiStepIndex].sTitle						:= 'DriveEnable On AllSubModules';
astAutoTable[udiStepIndex].udiModuleName				:= TPL.Gc_udiAllSubModules;
astAutoTable[udiStepIndex].diStep						:= diStep;
astAutoTable[udiStepIndex].diCmd						:= AXM.ET_Cmd.DriveEnableOn;
astAutoTable[udiStepIndex].timTimeOut					:= T#0MS;
astAutoTable[udiStepIndex].xEndCmd						:= FALSE;

TPL.FC_NextStep(udiStepIndex, diStep);
astAutoTable[udiStepIndex].sTitle						:= 'CamWs Mode AllSubModules';
astAutoTable[udiStepIndex].udiModuleName				:= TPL.Gc_udiAllSubModules;
astAutoTable[udiStepIndex].diStep						:= diStep;
astAutoTable[udiStepIndex].diCmd						:= AXM.ET_Cmd.CamWs;
astAutoTable[udiStepIndex].timTimeOut					:= T#0MS;
astAutoTable[udiStepIndex].xEndCmd						:= FALSE;

TPL.FC_NextStep(udiStepIndex, diStep);
astAutoTable[udiStepIndex].sTitle						:= 'Start AllSubModules';
astAutoTable[udiStepIndex].udiModuleName				:= TPL.Gc_udiAllSubModules;
astAutoTable[udiStepIndex].diStep						:= diStep;
astAutoTable[udiStepIndex].diCmd						:= AXM.ET_Cmd.Start;
astAutoTable[udiStepIndex].timTimeOut					:= T#0MS;
astAutoTable[udiStepIndex].xEndCmd						:= FALSE;

TPL.FC_NextStep(udiStepIndex, diStep);
astAutoTable[udiStepIndex].sTitle						:= 'WarmStart AllSubModules';
astAutoTable[udiStepIndex].udiModuleName				:= TPL.Gc_udiAllSubModules;
astAutoTable[udiStepIndex].diStep						:= diStep;
astAutoTable[udiStepIndex].diCmd						:= AXM.ET_Cmd.WsStart;
astAutoTable[udiStepIndex].timTimeOut					:= T#0MS;
astAutoTable[udiStepIndex].xEndCmd						:= FALSE;

TPL.FC_LastStep(udiStepIndex, diStep);
astAutoTable[udiStepIndex].sTitle						:= 'End';
astAutoTable[udiStepIndex].udiModuleName				:= 0;
astAutoTable[udiStepIndex].diStep						:= diStep;
astAutoTable[udiStepIndex].diCmd						:= 0;
astAutoTable[udiStepIndex].timTimeOut					:= T#0MS;
astAutoTable[udiStepIndex].xEndCmd						:= TRUE;

TPL.FC_NextCmdTable(iq_udiTableIndex:= udiTableIndex);
astListofCMDTables[udiTableIndex].sTitle				:= 'Auto';
astListofCMDTables[udiTableIndex].diCmd					:= ET_Cmd.Auto;
astListofCMDTables[udiTableIndex].udiNumberOfCmdSteps	:= udiStepIndex;

(*********************************************************************************************************************)
(*** Manual  ***)

TPL.FC_FirstStep(udiStepIndex, diStep);
astManualTable[udiStepIndex].sTitle						:= 'DriveEnable On AllSubModules';
astManualTable[udiStepIndex].udiModuleName				:= TPL.Gc_udiAllSubModules;
astManualTable[udiStepIndex].diStep						:= diStep;
astManualTable[udiStepIndex].diCmd						:= AXM.ET_Cmd.DriveEnableOn;
astManualTable[udiStepIndex].timTimeOut					:= T#0MS;
astManualTable[udiStepIndex].xEndCmd					:= FALSE;

TPL.FC_NextStep(udiStepIndex, diStep);
astManualTable[udiStepIndex].sTitle						:= 'Manual Mode AllSubModules';
astManualTable[udiStepIndex].udiModuleName				:= TPL.Gc_udiAllSubModules;
astManualTable[udiStepIndex].diStep						:= diStep;
astManualTable[udiStepIndex].diCmd						:= AXM.ET_Cmd.Manual;
astManualTable[udiStepIndex].timTimeOut					:= T#0MS;
astManualTable[udiStepIndex].xEndCmd					:= FALSE;

TPL.FC_LastStep(udiStepIndex, diStep);
astManualTable[udiStepIndex].sTitle						:= 'End';
astManualTable[udiStepIndex].udiModuleName				:= 0;
astManualTable[udiStepIndex].diStep						:= diStep;
astManualTable[udiStepIndex].diCmd						:= 0;
astManualTable[udiStepIndex].timTimeOut					:= T#0MS;
astManualTable[udiStepIndex].xEndCmd					:= TRUE;

TPL.FC_NextCmdTable(iq_udiTableIndex:= udiTableIndex);
astListofCMDTables[udiTableIndex].sTitle				:= 'Manual';
astListofCMDTables[udiTableIndex].diCmd					:= ET_Cmd.Manual;
astListofCMDTables[udiTableIndex].udiNumberOfCmdSteps	:= udiStepIndex;

(*********************************************************************************************************************)
(*** Stop ***)

TPL.FC_FirstStep(udiStepIndex, diStep);
astStopTable[udiStepIndex].sTitle						:= 'Stop AllSubModules';
astStopTable[udiStepIndex].udiModuleName				:= TPL.Gc_udiAllSubModules;
astStopTable[udiStepIndex].diStep						:= diStep;
astStopTable[udiStepIndex].diCmd						:= AXM.ET_Cmd.Stop;
astStopTable[udiStepIndex].timTimeOut					:= T#0MS;
astStopTable[udiStepIndex].xEndCmd						:= FALSE;

TPL.FC_LastStep(udiStepIndex, diStep);
astStopTable[udiStepIndex].sTitle						:= 'End';
astStopTable[udiStepIndex].udiModuleName				:= 0;
astStopTable[udiStepIndex].diStep						:= diStep;
astStopTable[udiStepIndex].diCmd						:= 0;
astStopTable[udiStepIndex].timTimeOut					:= T#0MS;
astStopTable[udiStepIndex].xEndCmd						:= TRUE;

TPL.FC_NextCmdTable(iq_udiTableIndex:= udiTableIndex);
astListofCMDTables[udiTableIndex].sTitle				:= 'Stop';
astListofCMDTables[udiTableIndex].diCmd					:= ET_Cmd.Stop;
astListofCMDTables[udiTableIndex].udiNumberOfCmdSteps	:= udiStepIndex;

(*********************************************************************************************************************)
(*** Start ***)

TPL.FC_FirstStep(udiStepIndex, diStep);
astStartTable[udiStepIndex].sTitle						:= 'Start AllSubModules';
astStartTable[udiStepIndex].udiModuleName				:= TPL.Gc_udiAllSubModules;
astStartTable[udiStepIndex].diStep						:= diStep;
astStartTable[udiStepIndex].diCmd						:= AXM.ET_Cmd.Start;
astStartTable[udiStepIndex].timTimeOut					:= T#0MS;
astStartTable[udiStepIndex].xEndCmd						:= FALSE;

TPL.FC_LastStep(udiStepIndex, diStep);
astStartTable[udiStepIndex].sTitle						:= 'End';
astStartTable[udiStepIndex].udiModuleName				:= 0;
astStartTable[udiStepIndex].diStep						:= diStep;
astStartTable[udiStepIndex].diCmd						:= 0;
astStartTable[udiStepIndex].timTimeOut					:= T#0MS;
astStartTable[udiStepIndex].xEndCmd						:= TRUE;

TPL.FC_NextCmdTable(iq_udiTableIndex:= udiTableIndex);
astListofCMDTables[udiTableIndex].sTitle				:= 'Start';
astListofCMDTables[udiTableIndex].diCmd					:= ET_Cmd.Start;
astListofCMDTables[udiTableIndex].udiNumberOfCmdSteps	:= udiStepIndex;

(*********************************************************************************************************************)
(*** Abort ***)

TPL.FC_FirstStep(udiStepIndex, diStep);
astAbortTable[udiStepIndex].sTitle						:= 'Stop AllSubModules';
astAbortTable[udiStepIndex].udiModuleName				:= TPL.Gc_udiAllSubModules;
astAbortTable[udiStepIndex].diStep						:= diStep;
astAbortTable[udiStepIndex].diCmd						:= AXM.ET_Cmd.Stop;
astAbortTable[udiStepIndex].timTimeOut					:= T#0MS;
astAbortTable[udiStepIndex].xEndCmd						:= FALSE;

TPL.FC_LastStep(udiStepIndex, diStep);
astAbortTable[udiStepIndex].sTitle						:= 'End';
astAbortTable[udiStepIndex].udiModuleName				:= 0;
astAbortTable[udiStepIndex].diStep						:= diStep;
astAbortTable[udiStepIndex].diCmd						:= 0;
astAbortTable[udiStepIndex].timTimeOut					:= T#0MS;
astAbortTable[udiStepIndex].xEndCmd						:= TRUE;

TPL.FC_NextCmdTable(iq_udiTableIndex:= udiTableIndex);
astListofCMDTables[udiTableIndex].sTitle				:= 'Abort';
astListofCMDTables[udiTableIndex].diCmd					:= ET_Cmd.Abort;
astListofCMDTables[udiTableIndex].udiNumberOfCmdSteps	:= udiStepIndex;

(*********************************************************************************************************************)
(*** Hold ***)

TPL.FC_FirstStep(udiStepIndex, diStep);
astHoldTable[udiStepIndex].sTitle						:= 'Hold AllSubModules';
astHoldTable[udiStepIndex].udiModuleName				:= TPL.Gc_udiAllSubModules;
astHoldTable[udiStepIndex].diStep						:= diStep;
astHoldTable[udiStepIndex].diCmd						:= AXM.ET_Cmd.Hold;
astHoldTable[udiStepIndex].timTimeOut					:= T#0MS;
astHoldTable[udiStepIndex].xEndCmd						:= FALSE;

TPL.FC_LastStep(udiStepIndex, diStep);
astHoldTable[udiStepIndex].sTitle						:= 'End';
astHoldTable[udiStepIndex].udiModuleName				:= 0;
astHoldTable[udiStepIndex].diStep						:= diStep;
astHoldTable[udiStepIndex].diCmd						:= 0;
astHoldTable[udiStepIndex].timTimeOut					:= T#0MS;
astHoldTable[udiStepIndex].xEndCmd						:= TRUE;

TPL.FC_NextCmdTable(iq_udiTableIndex:= udiTableIndex);
astListofCMDTables[udiTableIndex].sTitle				:= 'Hold';
astListofCMDTables[udiTableIndex].diCmd					:= ET_Cmd.Hold;
astListofCMDTables[udiTableIndex].udiNumberOfCmdSteps	:= udiStepIndex;

(*********************************************************************************************************************)
(*** Brake Release ***)

TPL.FC_FirstStep(udiStepIndex, diStep);
astBrakeReleaseTable[udiStepIndex].sTitle				:= 'DriveEnable Off AllSubModules';
astBrakeReleaseTable[udiStepIndex].udiModuleName		:= TPL.Gc_udiAllSubModules;
astBrakeReleaseTable[udiStepIndex].diStep				:= diStep;
astBrakeReleaseTable[udiStepIndex].diCmd				:= AXM.ET_Cmd.DriveEnableOff;
astBrakeReleaseTable[udiStepIndex].timTimeOut			:= T#0MS;
astBrakeReleaseTable[udiStepIndex].xEndCmd				:= FALSE;

TPL.FC_NextStep(udiStepIndex, diStep);
astBrakeReleaseTable[udiStepIndex].sTitle				:= 'BrakeRelease Mode AllSubModules';
astBrakeReleaseTable[udiStepIndex].udiModuleName		:= TPL.Gc_udiAllSubModules;
astBrakeReleaseTable[udiStepIndex].diStep				:= diStep;
astBrakeReleaseTable[udiStepIndex].diCmd				:= AXM.ET_Cmd.BrakeRelease;
astBrakeReleaseTable[udiStepIndex].timTimeOut			:= T#0MS;
astBrakeReleaseTable[udiStepIndex].xEndCmd				:= FALSE;

TPL.FC_NextStep(udiStepIndex, diStep);
astBrakeReleaseTable[udiStepIndex].sTitle				:= 'Start AllSubModules';
astBrakeReleaseTable[udiStepIndex].udiModuleName		:= TPL.Gc_udiAllSubModules;
astBrakeReleaseTable[udiStepIndex].diStep				:= diStep;
astBrakeReleaseTable[udiStepIndex].diCmd				:= AXM.ET_Cmd.Start;
astBrakeReleaseTable[udiStepIndex].timTimeOut			:= T#0MS;
astBrakeReleaseTable[udiStepIndex].xEndCmd				:= FALSE;

TPL.FC_LastStep(udiStepIndex, diStep);
astBrakeReleaseTable[udiStepIndex].sTitle				:= 'End';
astBrakeReleaseTable[udiStepIndex].udiModuleName		:= 0;
astBrakeReleaseTable[udiStepIndex].diStep				:= diStep;
astBrakeReleaseTable[udiStepIndex].diCmd				:= 0;
astBrakeReleaseTable[udiStepIndex].timTimeOut			:= T#0MS;
astBrakeReleaseTable[udiStepIndex].xEndCmd				:= TRUE;

TPL.FC_NextCmdTable(iq_udiTableIndex:= udiTableIndex);
astListofCMDTables[udiTableIndex].sTitle				:= 'BrakeRelease';
astListofCMDTables[udiTableIndex].diCmd					:= ET_Cmd.BrakeRelease;
astListofCMDTables[udiTableIndex].udiNumberOfCmdSteps	:= udiStepIndex;

(* End of system generated code, could be modified for your application *)
END_ACTION

ACTION Init_Exceptions:
(* System generated code, could be modified for your application *)
stUpdateStructsException.etDiag												:= GD.ET_Diag.UnexpectedProgramBehavior;
stUpdateStructsException.udiDiagExt											:= ET_DiagExt.UpdateStructsException;
stUpdateStructsException.sDiagExt											:= FC_EtDiagExtToString(i_etDiagExt := stUpdateStructsException.udiDiagExt);
stUpdateStructsException.sMsg												:= '';	(* Replaced on usage *)
stUpdateStructsException.udiModuleId										:= iq_stStandardModuleItf.i_udiModuleId;
stUpdateStructsException.sModuleName										:= iq_stStandardModuleItf.i_sModuleName;
stUpdateStructsException.stReaction.axReaction[TPL.ET_Reaction.AsyncStop]	:= TRUE;
stUpdateStructsException.etSource											:= TPL.ET_ExceptionSource.NodeModule;
stUpdateStructsException.timDelayTime										:= T#0MS;
stUpdateStructsException.wHmiAttributes										:= 0;
stUpdateStructsException.xAutoQuit											:= FALSE;

stInitReactionsException.etDiag												:= GD.ET_Diag.UnexpectedProgramBehavior;
stInitReactionsException.udiDiagExt											:= ET_DiagExt.InitReactionsException;
stInitReactionsException.sDiagExt											:= FC_EtDiagExtToString(i_etDiagExt := stInitReactionsException.udiDiagExt);
stInitReactionsException.sMsg												:= '';	(* Replaced on usage *)
stInitReactionsException.udiModuleId										:= iq_stStandardModuleItf.i_udiModuleId;
stInitReactionsException.sModuleName										:= iq_stStandardModuleItf.i_sModuleName;
stInitReactionsException.stReaction.axReaction[TPL.ET_Reaction.AsyncStop]	:= TRUE;
stInitReactionsException.etSource											:= TPL.ET_ExceptionSource.NodeModule;
stInitReactionsException.timDelayTime										:= T#0MS;
stInitReactionsException.wHmiAttributes										:= 0;
stInitReactionsException.xAutoQuit											:= FALSE;

stInitSubModulesException.etDiag											:= GD.ET_Diag.UnexpectedProgramBehavior;
stInitSubModulesException.udiDiagExt										:= ET_DiagExt.InitSubModulesException;
stInitSubModulesException.sDiagExt											:= FC_EtDiagExtToString(i_etDiagExt := stInitSubModulesException.udiDiagExt);
stInitSubModulesException.sMsg												:= '';	(* Replaced on usage *)
stInitSubModulesException.udiModuleId										:= iq_stStandardModuleItf.i_udiModuleId;
stInitSubModulesException.sModuleName										:= iq_stStandardModuleItf.i_sModuleName;
stInitSubModulesException.stReaction.axReaction[TPL.ET_Reaction.AsyncStop]	:= TRUE;
stInitSubModulesException.etSource											:= TPL.ET_ExceptionSource.NodeModule;
stInitSubModulesException.timDelayTime										:= T#0MS;
stInitSubModulesException.wHmiAttributes									:= 0;
stInitSubModulesException.xAutoQuit											:= FALSE;

		
(*------------------------------------------------------------------------------------------*)
(* Init User Exceptions *)

	// TPL.ET_Reaction.AsyncStop
	// TPL.ET_Reaction.SyncStopEL
	// TPL.ET_Reaction.SyncStopEH
	// TPL.ET_Reaction.StopEndOfCycle
	// TPL.ET_Reaction.MainsContactorOff

(*------------------------------------------------------------------------------------------*)
stUserException1.etDiag													:= GD.ET_Diag.ExecutionAborted;	 (* Replaced on usage *)
stUserException1.udiDiagExt												:= ET_DiagExtUser.Exception1FromEquipmentModule;	 (* Replaced on usage *)
stUserException1.sDiagExt												:= FC_EtDiagExtUserToString(i_etDiagExt := stUserException1.udiDiagExt);	 (* Replaced on usage *)
stUserException1.sMsg													:= 'User Exception 1';	 (* Replaced on usage *)
stUserException1.udiModuleId											:= iq_stStandardModuleItf.i_udiModuleId;
stUserException1.sModuleName											:= iq_stStandardModuleItf.i_sModuleName;
stUserException1.stReaction.axReaction[TPL.Gc_udiUserReactionOffset+2]	:= TRUE;
stUserException1.etSource												:= TPL.ET_ExceptionSource.User;
stUserException1.timDelayTime											:= T#0MS;
stUserException1.wHmiAttributes											:= 0;
stUserException1.xAutoQuit												:= FALSE;

stUserException2.etDiag													:= GD.ET_Diag.ExecutionAborted;	 (* Replaced on usage *)
stUserException2.udiDiagExt												:= ET_DiagExtUser.Exception2FromEquipmentModule;	 (* Replaced on usage *)
stUserException2.sDiagExt												:= FC_EtDiagExtUserToString(i_etDiagExt := stUserException2.udiDiagExt);	 (* Replaced on usage *)
stUserException2.sMsg													:= 'User Exception 2';	 (* Replaced on usage *)
stUserException2.udiModuleId											:= iq_stStandardModuleItf.i_udiModuleId;
stUserException2.sModuleName											:= iq_stStandardModuleItf.i_sModuleName;
stUserException2.stReaction.axReaction[TPL.Gc_udiUserReactionOffset+2]	:= TRUE;
stUserException2.etSource												:= TPL.ET_ExceptionSource.User;
stUserException2.timDelayTime											:= T#0MS;
stUserException2.wHmiAttributes											:= 0;
stUserException2.xAutoQuit												:= FALSE;

(* End of system generated code, could be modified for your application *)
END_ACTION

ACTION Init_Reactions:
(* System generated code, only to be changed by experienced programmers *)
IF c_udiNumberOfSubModules < 1 THEN
	RETURN;
END_IF

(* Change of default reactions only on demand *)
(* Compare SR MainMachine Action Init_Reactions *)

xInitReactionsException := FALSE;

(*****************************************************************************************************************************************************)
(* Init ReactionTranslationMode *)

TPL.FC_InitReactionTranslationMode(	i_udiNumberOfSubModules			:= c_udiNumberOfSubModules,
									i_petReactionTranslationMode	:= ADR(aetReactionTranslationMode),
									q_etDiag						=> etDiag,
									q_etDiagExt						=> etDiagExtTPL);
							
IF etDiag <> GD.ET_Diag.Ok AND NOT xInitReactionsException THEN
	xInitReactionsException := TRUE;
	
	stInitReactionsException.sMsg := PDL.FC_MultiConcat(i_sString1 := 'InitReactionTranslationMode - ', 
														i_sString2 := GD.FC_EtDiagToString(i_etDiag := etDiag), 
														i_sString3 := ' - ', 
														i_sString4 := TPL.FC_EtDiagExtToString(i_etDiagExt := etDiagExtTPL));
END_IF	

(*****************************************************************************************************************************************************)
(* Init ReactionTranslationTable *)	

TPL.FC_InitReactionTranslationTable(i_udiNumberOfSubModules			:= c_udiNumberOfSubModules,
									i_pstReactionTranslationTable	:= ADR(aastReactionTranslationTable),
									q_etDiag						=> etDiag,
									q_etDiagExt						=> etDiagExtTPL);
									
IF etDiag <> GD.ET_Diag.Ok AND NOT xInitReactionsException THEN
	xInitReactionsException := TRUE;
	
	stInitReactionsException.sMsg := PDL.FC_MultiConcat(i_sString1 := 'InitReactionTranslationTable - ', 
														i_sString2 := GD.FC_EtDiagToString(i_etDiag := etDiag), 
														i_sString3 := ' - ', 
														i_sString4 := TPL.FC_EtDiagExtToString(i_etDiagExt := etDiagExtTPL));
END_IF		

(*****************************************************************************************************************************************************)
(* Init ReactionTranslationJobs *)	
					
TPL.FC_InitReactionTranslationJobs( i_udiNumberOfSubModules			:= c_udiNumberOfSubModules,
									i_pstReactionTranslationJobs	:= ADR(astReactionTranslationJobs),
									q_etDiag						=> etDiag,
									q_etDiagExt						=> etDiagExtTPL);
						
IF etDiag <> GD.ET_Diag.Ok AND NOT xInitReactionsException THEN
	xInitReactionsException := TRUE;
	
	stInitReactionsException.sMsg := PDL.FC_MultiConcat(i_sString1 := 'InitReactionTranslationJobs - ', 
														i_sString2 := GD.FC_EtDiagToString(i_etDiag := etDiag), 
														i_sString3 := ' - ', 
														i_sString4 := TPL.FC_EtDiagExtToString(i_etDiagExt := etDiagExtTPL));
END_IF		

(*****************************************************************************************************************************************************)
(* Set exception if any exception occurred *)

TPL.FC_SetException(i_xExceptionActive	:= xInitReactionsException, 
					iq_stException		:= stInitReactionsException, 
					iq_stExceptionList	:= iq_stExceptionList, 
					iq_stLogDataList	:= iq_stLogDataList);
					
xInitSuccessful := xInitSuccessful AND NOT xInitReactionsException;

etDiag := GD.ET_Diag.Ok;
(* End of system generated code, only to be changed by experienced programmers *)
END_ACTION

ACTION Init_Slave1:
(* System generated code, could be modified for your application *)

(* Standard interface *)
astSubModuleInterface[c_udiSlave1].i_sModuleName		:= CONCAT(STR1 := iq_stStandardModuleItf.i_sModuleName, STR2 := ': Slave1');

astSubModuleInterface[c_udiSlave1].i_xLogEnable		:= 	TRUE;
astSubModuleInterface[c_udiSlave1].i_wLogDataFilter	:=	UDINT_TO_WORD(TPL.ET_LogDataFilter.ModuleDefault);

(* Axis main drive / EndlessFeed*)
stSlave1Interface.stMain.i_ifMaster		:= i_ifMaster; 		(* Master *)
stSlave1Interface.stMain.i_ifDrive		:= iq_stAdditionalItf.i_ifSlave1;
stSlave1Interface.stMain.iq_lencEncoder	:= iq_stAdditionalItf.i_lencEncoder1;


xDriveIsVirtual := FC_IsDriveVirtual(	i_ifDrive	:= stSlave1Interface.stMain.i_ifDrive,
										q_etDiag	=> etDiag,
										q_etDiagExt	=> etDiagExtTPL,
										q_sMsg		=> sMsgBuffer);

IF etDiag <> GD.ET_Diag.Ok AND NOT xIsDriveVirtualException THEN										
	stIsDriveVirtualException.sMsg := sMsgBuffer;
	xIsDriveVirtualException := TRUE;
END_IF

TPL.FC_SetException(i_xExceptionActive	:= xIsDriveVirtualException, 
					iq_stException		:= stIsDriveVirtualException, 
					iq_stExceptionList	:= iq_stExceptionList, 
					iq_stLogDataList	:= iq_stLogDataList);
					
xInitSuccessful := xInitSuccessful AND NOT xIsDriveVirtualException;
etDiag := GD.ET_Diag.Ok;
	

IF stSlave1Interface.stMain.i_ifMaster <> 0 THEN	
	stLogicalAddressMaster := stSlave1Interface.stMain.i_ifMaster.stLogicalAddress;
	IF (stLogicalAddressMaster.udiType = SYSTEMINTERFACE.P_ENC_TYPE.udiType) OR			(* Physical encoder *)
		(stLogicalAddressMaster.udiType = SYSTEMINTERFACE.INC_IN_TYPE.udiType) THEN		(* Incremental	encoder *)
		
		stLogicalAddressMaster.udiParameterId := 16#00A2;
		diResult := SYSTEMINTERFACE.FC_GetParameter(i_stLogAdr	:= stLogicalAddressMaster,
													i_dwBuffer	:= ADR(lrShaftRefDelay),
													i_diSize	:= SIZEOF(lrShaftRefDelay));
		IF diResult = 0 THEN
			stSlave1Interface.stMain.iq_lencEncoder.Delay := -lrShaftRefDelay;
		END_IF
	END_IF
END_IF


stSlave1Interface.stMain.i_lrMotionActiveVelLimit						:= 15.0;		(* Limit for max. velocity of astAxisModuleInterface to switch output AxisMove in Units/s *)
stSlave1Interface.stMain.i_etMotionActiveVelType						:= AXM.ET_MotionActiveVelType.Velocity;

stSlave1Interface.stMain.i_timMasterStop								:= T#1S;
stSlave1Interface.stMain.i_xHwLimitPos									:= FALSE;
stSlave1Interface.stMain.i_xHwLimitNeg									:= FALSE;

stSlave1Interface.stMain.stReducedVelocity.i_xEnableReducedVelocity		:= FALSE;
stSlave1Interface.stMain.stReducedVelocity.i_xOnlyLimitCheck			:= FALSE;
stSlave1Interface.stMain.stReducedVelocity.i_lrMaxReducedVelocity		:= 50.0;

stSlave1Interface.stMain.i_xStart										:= FALSE;

(***************************************************************************************************************************************************************************************************)

(*** Homing ***)

IF xDriveIsVirtual THEN
	stSlave1Interface.stHome.i_etMode := PDL.ET_HomeMode.SetPosAxisAndLogEncoderPosition;		(* Homing Mode in case of virtual axis *)
ELSE
	stSlave1Interface.stHome.i_etMode := PDL.ET_HomeMode.PosDirectionPosEdgeTp;					(* Homing Mode in case of real axis *)
END_IF


stSlave1Interface.stHome.i_xEnableInitAbsReadPos := TRUE;		(* TRUE : Restores the AxisPosition depending on the stHome.etMode
																		  If stHome.i_etMode is equal to PDL.ET_HomeMode.RestorePosFromAxisEncoder or 
																		  to PDL.ET_HomeMode.WriteAxisEncoder, the encoder of the axis is read,
																		  or else the position will be restored from the retain area *)

stSlave1Interface.stHome.stSetpos.iq_pstRestorePosRetain := iq_stAdditionalItf.i_pstRestorePosRetain1;

stSlave1Interface.stHome.i_xResetHomeOk := FALSE;

(* Possible modes for homing mode Sensor:
	PDL.ET_HomeMode.PosDirectionPosEdgeSensor
	PDL.ET_HomeMode.NegDirectionPosEdgeSensor
	PDL.ET_HomeMode.NegDirectionNegEdgeSensor
	PDL.ET_HomeMode.PosDirectionNegEdgeSensor
*)
stSlave1Interface.stHome.stSensor.i_lrHomePosition			:= 0.0;			(* Position at the end of homing in units *)
stSlave1Interface.stHome.stSensor.i_lrVel					:= 10.0;		(* Homing ceiling velocity in units/s *)
stSlave1Interface.stHome.stSensor.i_lrAcc					:= 1000.0;		(* Homing acceleration in units/s^2 *)
stSlave1Interface.stHome.stSensor.i_lrDec					:= 1000.0;		(* Homing deceleration in units/s^2 *)
stSlave1Interface.stHome.stSensor.i_lrJerk					:= 10000.0;		(* Homing jerk in units/s^3 *)
stSlave1Interface.stHome.stSensor.i_lrOffset				:= 0.0;			(* Offset from home signal in units *)
stSlave1Interface.stHome.stSensor.i_lrMaxTravel 			:= 720.0;		(* Max. travel for referencing by normal input *)
stSlave1Interface.stHome.stSensor.i_xRotativeSystem			:= FALSE;		(* Rotative system true or false for referencing by normal input *)
stSlave1Interface.stHome.stSensor.i_xSensor 				:= FALSE;		(* Input for home signal. Can be a signal from a controller input. Has to be written cyclic. *)

(* Possible Modes for homing mode LimitSwitch:
	PDL.ET_HomeMode.PosDirectionPosEdgeHWLimitPos		normally open contact / Closing contact
	PDL.ET_HomeMode.NegDirectionPosEdgeHWLimitNeg		normally open contact / Closing contact
	PDL.ET_HomeMode.NegDirectionNegEdgeHWLimitNeg		normally closed contact / Opening contact  
	PDL.ET_HomeMode.PosDirectionNegEdgeHWLimitPos		normally closed contact / Opening contact 
*)
stSlave1Interface.stHome.stLimitSwitch.i_lrHomePosition 	:= 0.0;			(* Position at the end of homing in units *)
stSlave1Interface.stHome.stLimitSwitch.i_lrVel				:= 10.0;		(* Homing ceiling velocity in units/s *)
stSlave1Interface.stHome.stLimitSwitch.i_lrLowVel			:= 5.0;			(* Homing low ceiling velocity in units/s *)
stSlave1Interface.stHome.stLimitSwitch.i_lrAcc				:= 1000.0;		(* Homing acceleration in units/s^2 *)
stSlave1Interface.stHome.stLimitSwitch.i_lrDec				:= 1000.0;		(* Homing deceleration in units/s^2 *)
stSlave1Interface.stHome.stLimitSwitch.i_lrJerk				:= 10000.0;		(* Homing jerk in units/s^3 *)
stSlave1Interface.stHome.stLimitSwitch.i_lrOffset			:= 0.0;			(* Offset from home signal in units *)
stSlave1Interface.stHome.stLimitSwitch.i_lrMaxTravel 		:= 9999.0;		(* Max. travel for referencing normal input as a hardware limit *)

(* Possible modes for homing mode MoveOnPos:
	PDL.ET_HomeMode.MoveOnPosAbs 
*)
stSlave1Interface.stHome.stMoveOnPos.i_lrTarget				:= 0.0;			(* Position at the end of homing in units *)
stSlave1Interface.stHome.stMoveOnPos.i_lrVel				:= 10.0;		(* Homing ceiling velocity in units/s *)
stSlave1Interface.stHome.stMoveOnPos.i_lrAcc				:= 1000.0;		(* Homing acceleration in units/s^2 *)
stSlave1Interface.stHome.stMoveOnPos.i_lrDec				:= 1000.0;		(* Homing deceleration in units/s^2 *)
stSlave1Interface.stHome.stMoveOnPos.i_lrJerk				:= 10000.0;		(* Homing jerk in units/s^3 *)
stSlave1Interface.stHome.stMoveOnPos.i_lrPeriod				:= 0.0;			(* Period of the axis *)
stSlave1Interface.stHome.stMoveOnPos.i_xRotativeSystem		:= FALSE;		(* Rotative system true or false *)

(* Possible modes for homing mode SetPos:
	PDL.ET_HomeMode.SetPosAxisPosition 
	PDL.ET_HomeMode.SetPosLogEncoderPosition 
	PDL.ET_HomeMode.SetPosAxisAndLogEncoderPosition
	PDL.ET_HomeMode.RestorePosFromAxisEncoder 
	PDL.ET_HomeMode.RestorePosFromRetain 
*)
stSlave1Interface.stHome.stSetpos.i_lrHomePosition			:= 0.0;			(* Position at the end of homing in units *)
stSlave1Interface.stHome.stSetpos.i_lrEncoderPosition		:= 0.0;			(* Encoder position in units after homing *)
stSlave1Interface.stHome.stSetpos.i_lrAbsEncOffset			:= 100.0;		(* Distance to the jump of axis encoder in units *)
stSlave1Interface.stHome.stSetpos.i_lrRestoreWindow			:= 180;			(* How far can the drive be away from its correct position *)
stSlave1Interface.stHome.stSetpos.i_lrUserPeriod			:= 360;			(* Period of the axis *)

(* Possible modes for homing mode Torque:
	PDL.ET_HomeMode.PosDirectionMaxTorque 
	PDL.ET_HomeMode.NegDirectionMaxTorque 
*)
stSlave1Interface.stHome.stTorque.i_lrHomePosition			:= 0.0;			(* Position at the end of homing in units *)
stSlave1Interface.stHome.stTorque.i_lrVel					:= 10.0;		(* Homing ceiling velocity in units/s *)
stSlave1Interface.stHome.stTorque.i_lrAcc					:= 1000.0;		(* Homing acceleration in units/s^2 *)
stSlave1Interface.stHome.stTorque.i_lrDec					:= 1000.0;		(* Homing deceleration in units/s^2 *)
stSlave1Interface.stHome.stTorque.i_lrJerk					:= 10000.0;		(* Homing jerk in units/s^3 *)
stSlave1Interface.stHome.stTorque.i_lrOffset				:= 0.0;			(* Offset from home signal in units *)
stSlave1Interface.stHome.stTorque.i_lrMaxTravel				:= 9999.0;		(* Max. travel for referencing by torque *)
stSlave1Interface.stHome.stTorque.i_lrMaxTorque				:= 0.0;			(* Torque for stop in Nm / referencing by torque *)
stSlave1Interface.stHome.stTorque.i_diTorqueTime			:= 5;			(* Time in msec to hold torque *)

(* Possible modes for homing mode TouchProbe:
	PDL.ET_HomeMode.PosDirectionPosEdgeTp 
	PDL.ET_HomeMode.NegDirectionPosEdgeTp 
	PDL.ET_HomeMode.NegDirectionNegEdgeTp 
	PDL.ET_HomeMode.PosDirectionNegEdgeTp 
*)
stSlave1Interface.stHome.stTouchProbe.i_lrHomePosition		:= 0.0;			(* Position at the end of homing in units *)
stSlave1Interface.stHome.stTouchProbe.i_lrVel				:= 100.0;		(* Homing ceiling velocity in units/s *)
stSlave1Interface.stHome.stTouchProbe.i_lrAcc				:= 1000.0;		(* Homing acceleration in units/s^2 *)
stSlave1Interface.stHome.stTouchProbe.i_lrDec				:= 1000.0;		(* Homing deceleration in units/s^2 *)
stSlave1Interface.stHome.stTouchProbe.i_lrJerk				:= 10000.0;		(* Homing jerk in units/s^3 *)
stSlave1Interface.stHome.stTouchProbe.i_lrOffset			:= 30.0;		(* Offset from home signal in units *)
stSlave1Interface.stHome.stTouchProbe.i_lrMaxTravel			:= 720.0;		(* Max. travel for referencing by TP *)
stSlave1Interface.stHome.stTouchProbe.i_xRotativeSystem		:= TRUE;		(* Rotative system true or false for referencing by TP *)
stSlave1Interface.stHome.stTouchProbe.i_ifTouchProbe		:= iq_stAdditionalItf.i_ifHomingTouchProbe1;		(* Input for TP *)

(* Possible modes for homing mode WritePos:
	PDL.ET_HomeMode.WriteAxisEncoder 
*)
stSlave1Interface.stHome.stWritePos.i_lrHomePosition		:= 0.0;			(* Position at the end of homing in units *)
stSlave1Interface.stHome.stWritePos.i_lrUserPeriod			:= 0.0;			(* Calculates Drive.Position into period ( units ) *)
stSlave1Interface.stHome.stWritePos.i_lrAbsEncOffset		:= 100.0;		(* Distance to the jump of axis encoder in units *)

(***************************************************************************************************************************************************************************************************)
(*** Manual ***)

stSlave1Interface.stManual.i_lrVel								:= 50.0;			(* Velocity in units/s *)
stSlave1Interface.stManual.i_lrAcc								:= 100.0;			(* Acceleration in units/s^2 *)
stSlave1Interface.stManual.i_lrDec								:= 100.0;			(* Deceleration in units/s^2 *)
stSlave1Interface.stManual.i_lrJerk								:= 1000.0;			(* Jerk in units/s^3 *)
stSlave1Interface.stManual.i_lrMaxDistance						:= 120.0;			(* Max pathlengths for one step in units *)
stSlave1Interface.stManual.i_xEndless							:= FALSE;			(* TRUE: jogging endless; Position between the periode; FALSE: jogging in steps. Position can be out of periode *)
stSlave1Interface.stManual.i_lrPeriod							:= 360.0;			(* Period of the axis *)

(***************************************************************************************************************************************************************************************************)
(*** Cam ***)

stSlave1Interface.stMultiCam.i_etCSModeSlave					:= PDL.ET_MultiCamCsModeSlave.SetSlavePositionToFirstCamPosition;		(* ColdStartMode Slave *)
stSlave1Interface.stMultiCam.i_etCSModeMaster					:= PDL.ET_MultiCamCsModeMaster.SetMasterPositionToFirstCamPosition;		(* ColdStartMode Master *)
stSlave1Interface.stMultiCam.i_etWSMode							:= PDL.ET_MultiCamWsMode.StoredCamMoveAlwaysNoPositionCheck;			(* WarmStartMode *)
stSlave1Interface.stMultiCam.i_lrWSWindow						:= 5.0;											(* WarmStartWindow in Axis units *)
stSlave1Interface.stMultiCam.i_lrWSVel							:= 10.0;										(* Velocity for WarmStart and CSModeSlave = PDL.ET_MultiCamCsModeSlave.MoveSlaveToFirstCamPosition in Units/s *)
stSlave1Interface.stMultiCam.i_lrWSAcc							:= 1000.0;										(* Acceleration and deceleration for Warmstart and CSModeSlave = PDL.ET_MultiCamCsModeSlave.MoveSlaveToFirstCamPosition in Units/s^2 *)
stSlave1Interface.stMultiCam.i_lrWSJerk							:= 10000.0;										(* Jerk for Warmstart and CSModeSlave = PDL.ET_MultiCamCsModeSlave.MoveSlaveToFirstCamPosition in units/s^3 *)
stSlave1Interface.stMultiCam.i_diTXend							:= 2*SYSTEMINTERFACE.FC_LzsTaskGetInterval();	(* Time of XLowEnd and XHighEnd befor Xend or Xstart in msec*)
stSlave1Interface.stMultiCam.i_lrInstantXLimMax					:= 0.0;											(* Switch off position at 'InstantNewCam' *)

stSlave1Interface.stMultiCam.i_xEnableTabHandler				:= TRUE;										(* TRUE: TabHandler is enabled *)
stSlave1Interface.stMultiCam.i_udiTableSelectNr					:= AXM.ET_ParId.User;							(* Number of table which is used in the next cycle *)								

stSlave1Interface.stMultiCam.i_xSetEncoderParameters			:= FALSE;										(* TRUE: The parameters MasterId, FeedConstand, GearIn and GearOut will be copyed into LEnc object *)
stSlave1Interface.stMultiCam.i_xSetEncoderPosition				:= FALSE;										(* TRUE: Manipulation of LEnc object on startup OpMode MultiCam *)
stSlave1Interface.stMultiCam.i_lrSetEncoderOffset				:= 0.0;											(* Master encoder offset *)
stSlave1Interface.stMultiCam.i_xCheckEncoderPeriod				:= TRUE;										(* TRUE: Check of encoder period = 0. If encoder period <> 0 -> Exception *)

stSlave1Interface.stMultiCam.iq_astMotionPar[AXM.ET_ParId.User].diNumberOfCamPoints			:= 4;	(* DataStruct for the next cycle *)
stSlave1Interface.stMultiCam.iq_astMotionPar[AXM.ET_ParId.User].lrYPeriod						:= 0.0;

stSlave1Interface.stMultiCam.iq_astMotionPar[AXM.ET_ParId.User].astCamPoint[0].lrX			:= 0.0;
stSlave1Interface.stMultiCam.iq_astMotionPar[AXM.ET_ParId.User].astCamPoint[0].lrY			:= 0.0;
stSlave1Interface.stMultiCam.iq_astMotionPar[AXM.ET_ParId.User].astCamPoint[0].lrM			:= 0.0;
stSlave1Interface.stMultiCam.iq_astMotionPar[AXM.ET_ParId.User].astCamPoint[0].etCamType	:= PDL.ET_CamType.Poly5Com;
stSlave1Interface.stMultiCam.iq_astMotionPar[AXM.ET_ParId.User].astCamPoint[1].lrX			:= 60.0;
stSlave1Interface.stMultiCam.iq_astMotionPar[AXM.ET_ParId.User].astCamPoint[1].lrY			:= 30.0;
stSlave1Interface.stMultiCam.iq_astMotionPar[AXM.ET_ParId.User].astCamPoint[1].lrM			:= 1.0;
stSlave1Interface.stMultiCam.iq_astMotionPar[AXM.ET_ParId.User].astCamPoint[1].etCamType	:= PDL.ET_CamType.Straight;
stSlave1Interface.stMultiCam.iq_astMotionPar[AXM.ET_ParId.User].astCamPoint[2].lrX			:= 240.0;
stSlave1Interface.stMultiCam.iq_astMotionPar[AXM.ET_ParId.User].astCamPoint[2].lrY			:= 210.0;
stSlave1Interface.stMultiCam.iq_astMotionPar[AXM.ET_ParId.User].astCamPoint[2].lrM			:= 1.0;
stSlave1Interface.stMultiCam.iq_astMotionPar[AXM.ET_ParId.User].astCamPoint[2].etCamType	:= PDL.ET_CamType.Poly5Com;
stSlave1Interface.stMultiCam.iq_astMotionPar[AXM.ET_ParId.User].astCamPoint[3].lrX			:= 360.0;
stSlave1Interface.stMultiCam.iq_astMotionPar[AXM.ET_ParId.User].astCamPoint[3].lrY			:= 0.0;
stSlave1Interface.stMultiCam.iq_astMotionPar[AXM.ET_ParId.User].astCamPoint[3].lrM			:= 0.0;
stSlave1Interface.stMultiCam.iq_astMotionPar[AXM.ET_ParId.User].astCamPoint[3].etCamType	:= PDL.ET_CamType.Poly5Com;

stSlave1Interface.stMultiCam.iq_astMotionPar[AXM.ET_ParId.Idle].diUserTableId	:= AXM.ET_ParId.Idle;
stSlave1Interface.stMultiCam.iq_astMotionPar[AXM.ET_ParId.Start].diUserTableId	:= AXM.ET_ParId.Start;
stSlave1Interface.stMultiCam.iq_astMotionPar[AXM.ET_ParId.Cont].diUserTableId	:= AXM.ET_ParId.Cont;
stSlave1Interface.stMultiCam.iq_astMotionPar[AXM.ET_ParId.Stop].diUserTableId	:= AXM.ET_ParId.Stop;
stSlave1Interface.stMultiCam.iq_astMotionPar[AXM.ET_ParId.User].diUserTableId	:= AXM.ET_ParId.User;


(***************************************************************************************************************************************************************************************************)
(*** Endless ***)

stSlave1Interface.stEndless.i_lrVel								:= 100.0;			(* Velocity in Units/s *)
stSlave1Interface.stEndless.i_lrAcc								:= 1000.0;			(* Acceleration in Units/s^2 *)
stSlave1Interface.stEndless.i_lrDec								:= 1000.0;			(* Deceleration in Units/s^2 *)
stSlave1Interface.stEndless.i_lrJerk							:= 10000.0;			(* Jerk in units/s^3 *)
stSlave1Interface.stEndless.i_lrPeriod							:= 360.0;			(* Period one cycle in units *)
stSlave1Interface.stEndless.i_lrStopPosition					:= 0.5;				(* Stop position in units *)


(***************************************************************************************************************************************************************************************************)
(*** Pos ***)

stSlave1Interface.stPos.i_etPosMode								:= SYSTEMINTERFACE.ET_PosMode.Endless;		(* SYSTEMINTERFACE.ET_PosMode.Endless, SYSTEMINTERFACE.ET_PosMode.Relative, SYSTEMINTERFACE.ET_PosMode.Absolute *)
stSlave1Interface.stPos.i_lrTarget								:= 360.0;									(* Target position or distance in Units *)
stSlave1Interface.stPos.i_lrVel									:= 360.0;									(* Ceiling velocity in Units/s *)
stSlave1Interface.stPos.i_lrAcc									:= 3600.0;									(* Acceleration in Units/s^2 *)
stSlave1Interface.stPos.i_lrDec									:= 3600.0;									(* Deceleration in Units/s^2 *)
stSlave1Interface.stPos.i_lrJerk								:= 36000.0;									(* Jerk in units/s^3 *)


(* End of system generated code, could be modified for your application *)
END_ACTION

ACTION Init_Slave2:
(* System generated code, could be modified for your application *)

(* Standard interface *)
astSubModuleInterface[c_udiSlave2].i_sModuleName		:= CONCAT(STR1 := iq_stStandardModuleItf.i_sModuleName, STR2 := ': Slave2');

astSubModuleInterface[c_udiSlave2].i_xLogEnable		:= 	TRUE;
astSubModuleInterface[c_udiSlave2].i_wLogDataFilter	:= 	UDINT_TO_WORD(TPL.ET_LogDataFilter.ModuleDefault);

(* Axis main drive / EndlessFeed*)
stSlave2Interface.stMain.i_ifMaster		:= i_ifMaster; 		(* Master *)
stSlave2Interface.stMain.i_ifDrive 		:= iq_stAdditionalItf.i_ifSlave2;
stSlave2Interface.stMain.iq_lencEncoder	:= iq_stAdditionalItf.i_lencEncoder2;


xDriveIsVirtual := FC_IsDriveVirtual(	i_ifDrive	:= stSlave2Interface.stMain.i_ifDrive,
										q_etDiag	=> etDiag,
										q_etDiagExt	=> etDiagExtTPL,
										q_sMsg		=> sMsgBuffer);

IF etDiag <> GD.ET_Diag.Ok AND NOT xIsDriveVirtualException THEN										
	stIsDriveVirtualException.sMsg := sMsgBuffer;
	xIsDriveVirtualException := TRUE;
END_IF

TPL.FC_SetException(i_xExceptionActive	:= xIsDriveVirtualException, 
					iq_stException		:= stIsDriveVirtualException, 
					iq_stExceptionList	:= iq_stExceptionList, 
					iq_stLogDataList	:= iq_stLogDataList);
					
xInitSuccessful := xInitSuccessful AND NOT xIsDriveVirtualException;
etDiag := GD.ET_Diag.Ok;
	

IF stSlave2Interface.stMain.i_ifMaster <> 0 THEN	
	stLogicalAddressMaster := stSlave2Interface.stMain.i_ifMaster.stLogicalAddress;
	IF (stLogicalAddressMaster.udiType = SYSTEMINTERFACE.P_ENC_TYPE.udiType) OR			(* Physical encoder *)
		(stLogicalAddressMaster.udiType = SYSTEMINTERFACE.INC_IN_TYPE.udiType) THEN		(* Incremental	encoder *)
		
		stLogicalAddressMaster.udiParameterId := 16#00A2;
		diResult := SYSTEMINTERFACE.FC_GetParameter(i_stLogAdr	:= stLogicalAddressMaster,
													i_dwBuffer	:= ADR(lrShaftRefDelay),
													i_diSize	:= SIZEOF(lrShaftRefDelay));
		IF diResult = 0 THEN
			stSlave2Interface.stMain.iq_lencEncoder.Delay := -lrShaftRefDelay;
		END_IF
	END_IF
END_IF


stSlave2Interface.stMain.i_lrMotionActiveVelLimit						:= 15.0;		(* Limit for max. velocity of astAxisModuleInterface to switch output AxisMove in Units/s *)
stSlave2Interface.stMain.i_etMotionActiveVelType						:= AXM.ET_MotionActiveVelType.Velocity;

stSlave2Interface.stMain.i_timMasterStop								:= T#1S;
stSlave2Interface.stMain.i_xHwLimitPos									:= FALSE;
stSlave2Interface.stMain.i_xHwLimitNeg									:= FALSE;

stSlave2Interface.stMain.stReducedVelocity.i_xEnableReducedVelocity		:= FALSE;
stSlave2Interface.stMain.stReducedVelocity.i_xOnlyLimitCheck			:= FALSE;
stSlave2Interface.stMain.stReducedVelocity.i_lrMaxReducedVelocity		:= 50.0;

stSlave2Interface.stMain.i_xStart										:= FALSE;

(***************************************************************************************************************************************************************************************************)

(*** Homing ***)

IF xDriveIsVirtual THEN
	stSlave2Interface.stHome.i_etMode := PDL.ET_HomeMode.SetPosAxisAndLogEncoderPosition;		(* Homing Mode in case of virtual axis *)
ELSE
	stSlave2Interface.stHome.i_etMode := PDL.ET_HomeMode.SetPosAxisAndLogEncoderPosition;		(* Homing Mode in case of real axis *)
END_IF


stSlave2Interface.stHome.i_xEnableInitAbsReadPos := TRUE;		(* TRUE : Restores the AxisPosition depending on the stHome.etMode
																		  If stHome.i_etMode is equal to PDL.ET_HomeMode.RestorePosFromAxisEncoder or 
																		  to PDL.ET_HomeMode.WriteAxisEncoder, the encoder of the axis is read,
																		  or else the position will be restored from the retain area *)

stSlave2Interface.stHome.stSetpos.iq_pstRestorePosRetain := iq_stAdditionalItf.i_pstRestorePosRetain2;

stSlave2Interface.stHome.i_xResetHomeOk := FALSE;

(* Possible modes for homing mode Sensor:
	PDL.ET_HomeMode.PosDirectionPosEdgeSensor
	PDL.ET_HomeMode.NegDirectionPosEdgeSensor
	PDL.ET_HomeMode.NegDirectionNegEdgeSensor
	PDL.ET_HomeMode.PosDirectionNegEdgeSensor
*)
stSlave2Interface.stHome.stSensor.i_lrHomePosition			:= 0.0;			(* Position at the end of homing in units *)
stSlave2Interface.stHome.stSensor.i_lrVel					:= 10.0;		(* Homing ceiling velocity in units/s *)
stSlave2Interface.stHome.stSensor.i_lrAcc					:= 1000.0;		(* Homing acceleration in units/s^2 *)
stSlave2Interface.stHome.stSensor.i_lrDec					:= 1000.0;		(* Homing deceleration in units/s^2 *)
stSlave2Interface.stHome.stSensor.i_lrJerk					:= 10000.0;		(* Homing jerk in units/s^3 *)
stSlave2Interface.stHome.stSensor.i_lrOffset				:= 0.0;			(* Offset from home signal in units *)
stSlave2Interface.stHome.stSensor.i_lrMaxTravel 			:= 720.0;		(* Max. travel for referencing by normal input *)
stSlave2Interface.stHome.stSensor.i_xRotativeSystem			:= FALSE;		(* Rotative system true or false for referencing by normal input *)
stSlave2Interface.stHome.stSensor.i_xSensor 				:= FALSE;		(* Input for home signal. Can be a signal from a controller input. Has to be written cyclic. *)

(* Possible Modes for homing mode LimitSwitch:
	PDL.ET_HomeMode.PosDirectionPosEdgeHWLimitPos		normally open contact / Closing contact
	PDL.ET_HomeMode.NegDirectionPosEdgeHWLimitNeg		normally open contact / Closing contact
	PDL.ET_HomeMode.NegDirectionNegEdgeHWLimitNeg		normally closed contact / Opening contact  
	PDL.ET_HomeMode.PosDirectionNegEdgeHWLimitPos		normally closed contact / Opening contact 
*)
stSlave2Interface.stHome.stLimitSwitch.i_lrHomePosition 	:= 0.0;			(* Position at the end of homing in units *)
stSlave2Interface.stHome.stLimitSwitch.i_lrVel				:= 10.0;		(* Homing ceiling velocity in units/s *)
stSlave2Interface.stHome.stLimitSwitch.i_lrLowVel			:= 5.0;			(* Homing low ceiling velocity in units/s *)
stSlave2Interface.stHome.stLimitSwitch.i_lrAcc				:= 1000.0;		(* Homing acceleration in units/s^2 *)
stSlave2Interface.stHome.stLimitSwitch.i_lrDec				:= 1000.0;		(* Homing deceleration in units/s^2 *)
stSlave2Interface.stHome.stLimitSwitch.i_lrJerk				:= 10000.0;		(* Homing jerk in units/s^3 *)
stSlave2Interface.stHome.stLimitSwitch.i_lrOffset			:= 0.0;			(* Offset from home signal in units *)
stSlave2Interface.stHome.stLimitSwitch.i_lrMaxTravel 		:= 9999.0;		(* Max. travel for referencing normal input as a hardware limit *)

(* Possible modes for homing mode MoveOnPos:
	PDL.ET_HomeMode.MoveOnPosAbs 
*)
stSlave2Interface.stHome.stMoveOnPos.i_lrTarget				:= 0.0;			(* Position at the end of homing in units *)
stSlave2Interface.stHome.stMoveOnPos.i_lrVel				:= 10.0;		(* Homing ceiling velocity in units/s *)
stSlave2Interface.stHome.stMoveOnPos.i_lrAcc				:= 1000.0;		(* Homing acceleration in units/s^2 *)
stSlave2Interface.stHome.stMoveOnPos.i_lrDec				:= 1000.0;		(* Homing deceleration in units/s^2 *)
stSlave2Interface.stHome.stMoveOnPos.i_lrJerk				:= 10000.0;		(* Homing jerk in units/s^3 *)
stSlave2Interface.stHome.stMoveOnPos.i_lrPeriod				:= 0.0;			(* Period of the axis *)
stSlave2Interface.stHome.stMoveOnPos.i_xRotativeSystem		:= FALSE;		(* Rotative system true or false *)

(* Possible modes for homing mode SetPos:
	PDL.ET_HomeMode.SetPosAxisPosition 
	PDL.ET_HomeMode.SetPosLogEncoderPosition 
	PDL.ET_HomeMode.SetPosAxisAndLogEncoderPosition
	PDL.ET_HomeMode.RestorePosFromAxisEncoder 
	PDL.ET_HomeMode.RestorePosFromRetain 
*)
stSlave2Interface.stHome.stSetpos.i_lrHomePosition			:= 0.0;			(* Position at the end of homing in units *)
stSlave2Interface.stHome.stSetpos.i_lrEncoderPosition		:= 0.0;			(* Encoder position in units after homing *)
stSlave2Interface.stHome.stSetpos.i_lrAbsEncOffset			:= 100.0;		(* Distance to the jump of axis encoder in units *)
stSlave2Interface.stHome.stSetpos.i_lrRestoreWindow			:= 180;			(* How far can the drive be away from its correct position *)
stSlave2Interface.stHome.stSetpos.i_lrUserPeriod			:= 360;			(* Period of the axis *)

(* Possible modes for homing mode Torque:
	PDL.ET_HomeMode.PosDirectionMaxTorque 
	PDL.ET_HomeMode.NegDirectionMaxTorque 
*)
stSlave2Interface.stHome.stTorque.i_lrHomePosition			:= 0.0;			(* Position at the end of homing in units *)
stSlave2Interface.stHome.stTorque.i_lrVel					:= 10.0;		(* Homing ceiling velocity in units/s *)
stSlave2Interface.stHome.stTorque.i_lrAcc					:= 1000.0;		(* Homing acceleration in units/s^2 *)
stSlave2Interface.stHome.stTorque.i_lrDec					:= 1000.0;		(* Homing deceleration in units/s^2 *)
stSlave2Interface.stHome.stTorque.i_lrJerk					:= 10000.0;		(* Homing jerk in units/s^3 *)
stSlave2Interface.stHome.stTorque.i_lrOffset				:= 0.0;			(* Offset from home signal in units *)
stSlave2Interface.stHome.stTorque.i_lrMaxTravel				:= 9999.0;		(* Max. travel for referencing by torque *)
stSlave2Interface.stHome.stTorque.i_lrMaxTorque				:= 0.0;			(* Torque for stop in Nm / referencing by torque *)
stSlave2Interface.stHome.stTorque.i_diTorqueTime			:= 5;			(* Time in msec to hold torque *)

(* Possible modes for homing mode TouchProbe:
	PDL.ET_HomeMode.PosDirectionPosEdgeTp 
	PDL.ET_HomeMode.NegDirectionPosEdgeTp 
	PDL.ET_HomeMode.NegDirectionNegEdgeTp 
	PDL.ET_HomeMode.PosDirectionNegEdgeTp 
*)
stSlave2Interface.stHome.stTouchProbe.i_lrHomePosition		:= 0.0;			(* Position at the end of homing in units *)
stSlave2Interface.stHome.stTouchProbe.i_lrVel				:= 100.0;		(* Homing ceiling velocity in units/s *)
stSlave2Interface.stHome.stTouchProbe.i_lrAcc				:= 1000.0;		(* Homing acceleration in units/s^2 *)
stSlave2Interface.stHome.stTouchProbe.i_lrDec				:= 1000.0;		(* Homing deceleration in units/s^2 *)
stSlave2Interface.stHome.stTouchProbe.i_lrJerk				:= 10000.0;		(* Homing jerk in units/s^3 *)
stSlave2Interface.stHome.stTouchProbe.i_lrOffset			:= 30.0;		(* Offset from home signal in units *)
stSlave2Interface.stHome.stTouchProbe.i_lrMaxTravel			:= 720.0;		(* Max. travel for referencing by TP *)
stSlave2Interface.stHome.stTouchProbe.i_xRotativeSystem		:= TRUE;		(* Rotative system true or false for referencing by TP *)
stSlave2Interface.stHome.stTouchProbe.i_ifTouchProbe		:= iq_stAdditionalItf.i_ifHomingTouchProbe2;		(* Input for TP *)

(* Possible modes for homing mode WritePos:
	PDL.ET_HomeMode.WriteAxisEncoder 
*)
stSlave2Interface.stHome.stWritePos.i_lrHomePosition		:= 0.0;			(* Position at the end of homing in units *)
stSlave2Interface.stHome.stWritePos.i_lrUserPeriod			:= 0.0;			(* Calculates Drive.Position into period ( units ) *)
stSlave2Interface.stHome.stWritePos.i_lrAbsEncOffset		:= 100.0;		(* Distance to the jump of axis encoder in units *)

(***************************************************************************************************************************************************************************************************)
(*** Manual ***)

stSlave2Interface.stManual.i_lrVel								:= 50.0;			(* Velocity in units/s *)
stSlave2Interface.stManual.i_lrAcc								:= 100.0;			(* Acceleration in units/s^2 *)
stSlave2Interface.stManual.i_lrDec								:= 100.0;			(* Deceleration in units/s^2 *)
stSlave2Interface.stManual.i_lrJerk								:= 1000.0;			(* Jerk in units/s^3 *)
stSlave2Interface.stManual.i_lrMaxDistance						:= 120.0;			(* Max pathlengths for one step in units *)
stSlave2Interface.stManual.i_xEndless							:= FALSE;			(* TRUE: jogging endless; Position between the periode; FALSE: jogging in steps. Position can be out of periode *)
stSlave2Interface.stManual.i_lrPeriod							:= 360.0;			(* Period of the axis *)

(***************************************************************************************************************************************************************************************************)
(*** Cam ***)

stSlave2Interface.stMultiCam.i_etCSModeSlave					:= PDL.ET_MultiCamCsModeSlave.SetSlavePositionToFirstCamPosition;		(* ColdStartMode Slave *)
stSlave2Interface.stMultiCam.i_etCSModeMaster					:= PDL.ET_MultiCamCsModeMaster.SetMasterPositionToFirstCamPosition;		(* ColdStartMode Master *)
stSlave2Interface.stMultiCam.i_etWSMode							:= PDL.ET_MultiCamWsMode.StoredCamMoveAlwaysNoPositionCheck;			(* WarmStartMode *)
stSlave2Interface.stMultiCam.i_lrWSWindow						:= 5.0;											(* WarmStartWindow in Axis units *)
stSlave2Interface.stMultiCam.i_lrWSVel							:= 10.0;										(* Velocity for WarmStart and CSModeSlave = PDL.ET_MultiCamCsModeSlave.MoveSlaveToFirstCamPosition in Units/s *)
stSlave2Interface.stMultiCam.i_lrWSAcc							:= 1000.0;										(* Acceleration and deceleration for Warmstart and CSModeSlave = PDL.ET_MultiCamCsModeSlave.MoveSlaveToFirstCamPosition in Units/s^2 *)
stSlave2Interface.stMultiCam.i_lrWSJerk							:= 10000.0;										(* Jerk for Warmstart and CSModeSlave = PDL.ET_MultiCamCsModeSlave.MoveSlaveToFirstCamPosition in units/s^3 *)
stSlave2Interface.stMultiCam.i_diTXend							:= 2*SYSTEMINTERFACE.FC_LzsTaskGetInterval();	(* Time of XLowEnd and XHighEnd befor Xend or Xstart in msec*)
stSlave2Interface.stMultiCam.i_lrInstantXLimMax					:= 0.0;											(* Switch off position at 'InstantNewCam' *)

stSlave2Interface.stMultiCam.i_xEnableTabHandler				:= TRUE;										(* TRUE: TabHandler is enabled *)
stSlave2Interface.stMultiCam.i_udiTableSelectNr					:= AXM.ET_ParId.User;							(* Number of table which is used in the next cycle *)								

stSlave2Interface.stMultiCam.i_xSetEncoderParameters			:= FALSE;										(* TRUE: The parameters MasterId, FeedConstand, GearIn and GearOut will be copyed into LEnc object *)
stSlave2Interface.stMultiCam.i_xSetEncoderPosition				:= FALSE;										(* TRUE: Manipulation of LEnc object on startup OpMode MultiCam *)
stSlave2Interface.stMultiCam.i_lrSetEncoderOffset				:= 0.0;											(* Master encoder offset *)
stSlave2Interface.stMultiCam.i_xCheckEncoderPeriod				:= TRUE;										(* TRUE: Check of encoder period = 0. If encoder period <> 0 -> Exception *)

stSlave2Interface.stMultiCam.iq_astMotionPar[AXM.ET_ParId.User].diNumberOfCamPoints			:= 4;	(* DataStruct for the next cycle *)
stSlave2Interface.stMultiCam.iq_astMotionPar[AXM.ET_ParId.User].lrYPeriod						:= 0.0;

stSlave2Interface.stMultiCam.iq_astMotionPar[AXM.ET_ParId.User].astCamPoint[0].lrX			:= 0.0;
stSlave2Interface.stMultiCam.iq_astMotionPar[AXM.ET_ParId.User].astCamPoint[0].lrY			:= 0.0;
stSlave2Interface.stMultiCam.iq_astMotionPar[AXM.ET_ParId.User].astCamPoint[0].lrM			:= 0.0;
stSlave2Interface.stMultiCam.iq_astMotionPar[AXM.ET_ParId.User].astCamPoint[0].etCamType	:= PDL.ET_CamType.Poly5Com;
stSlave2Interface.stMultiCam.iq_astMotionPar[AXM.ET_ParId.User].astCamPoint[1].lrX			:= 60.0;
stSlave2Interface.stMultiCam.iq_astMotionPar[AXM.ET_ParId.User].astCamPoint[1].lrY			:= 30.0;
stSlave2Interface.stMultiCam.iq_astMotionPar[AXM.ET_ParId.User].astCamPoint[1].lrM			:= 1.0;
stSlave2Interface.stMultiCam.iq_astMotionPar[AXM.ET_ParId.User].astCamPoint[1].etCamType	:= PDL.ET_CamType.Straight;
stSlave2Interface.stMultiCam.iq_astMotionPar[AXM.ET_ParId.User].astCamPoint[2].lrX			:= 240.0;
stSlave2Interface.stMultiCam.iq_astMotionPar[AXM.ET_ParId.User].astCamPoint[2].lrY			:= 210.0;
stSlave2Interface.stMultiCam.iq_astMotionPar[AXM.ET_ParId.User].astCamPoint[2].lrM			:= 1.0;
stSlave2Interface.stMultiCam.iq_astMotionPar[AXM.ET_ParId.User].astCamPoint[2].etCamType	:= PDL.ET_CamType.Poly5Com;
stSlave2Interface.stMultiCam.iq_astMotionPar[AXM.ET_ParId.User].astCamPoint[3].lrX			:= 360.0;
stSlave2Interface.stMultiCam.iq_astMotionPar[AXM.ET_ParId.User].astCamPoint[3].lrY			:= 0.0;
stSlave2Interface.stMultiCam.iq_astMotionPar[AXM.ET_ParId.User].astCamPoint[3].lrM			:= 0.0;
stSlave2Interface.stMultiCam.iq_astMotionPar[AXM.ET_ParId.User].astCamPoint[3].etCamType	:= PDL.ET_CamType.Poly5Com;

stSlave2Interface.stMultiCam.iq_astMotionPar[AXM.ET_ParId.Idle].diUserTableId	:= AXM.ET_ParId.Idle;
stSlave2Interface.stMultiCam.iq_astMotionPar[AXM.ET_ParId.Start].diUserTableId	:= AXM.ET_ParId.Start;
stSlave2Interface.stMultiCam.iq_astMotionPar[AXM.ET_ParId.Cont].diUserTableId	:= AXM.ET_ParId.Cont;
stSlave2Interface.stMultiCam.iq_astMotionPar[AXM.ET_ParId.Stop].diUserTableId	:= AXM.ET_ParId.Stop;
stSlave2Interface.stMultiCam.iq_astMotionPar[AXM.ET_ParId.User].diUserTableId	:= AXM.ET_ParId.User;



(***************************************************************************************************************************************************************************************************)
(*** Endless ***)

stSlave2Interface.stEndless.i_lrVel								:= 100.0;			(* Velocity in Units/s *)
stSlave2Interface.stEndless.i_lrAcc								:= 1000.0;			(* Acceleration in Units/s^2 *)
stSlave2Interface.stEndless.i_lrDec								:= 1000.0;			(* Deceleration in Units/s^2 *)
stSlave2Interface.stEndless.i_lrJerk							:= 10000.0;			(* Jerk in units/s^3 *)
stSlave2Interface.stEndless.i_lrPeriod							:= 360.0;			(* Period one cycle in units *)
stSlave2Interface.stEndless.i_lrStopPosition					:= 0.5;				(* Stop position in units *)



(***************************************************************************************************************************************************************************************************)
(*** Pos ***)

stSlave2Interface.stPos.i_etPosMode								:= SYSTEMINTERFACE.ET_PosMode.Endless;		(* SYSTEMINTERFACE.ET_PosMode.Endless, SYSTEMINTERFACE.ET_PosMode.Relative, SYSTEMINTERFACE.ET_PosMode.Absolute *)
stSlave2Interface.stPos.i_lrTarget								:= 360.0;									(* Target position or distance in Units *)
stSlave2Interface.stPos.i_lrVel									:= 360.0;									(* Ceiling velocity in Units/s *)
stSlave2Interface.stPos.i_lrAcc									:= 3600.0;									(* Acceleration in Units/s^2 *)
stSlave2Interface.stPos.i_lrDec									:= 3600.0;									(* Deceleration in Units/s^2 *)
stSlave2Interface.stPos.i_lrJerk								:= 36000.0;									(* Jerk in units/s^3 *)


(* End of system generated code, could be modified for your application *)
END_ACTION

ACTION Init_SubModules:
(* System generated code, could be modified for your application *)

(* Module Group declaration *)

aaudiSubModuleGroups[c_udiSlaveGroup1-TPL.Gc_udiGroupOffset,TPL.ET_Group.Member1]	:= 0;			(* There is no first element of the group c_udiSlaveGroup1 *)
aaudiSubModuleGroups[c_udiSlaveGroup1-TPL.Gc_udiGroupOffset,TPL.ET_Group.Member2]	:= 0;			(* There is no second element of the group c_udiSlaveGroup1 *)

aaudiSubModuleGroups[c_udiSlaveGroup2-TPL.Gc_udiGroupOffset,TPL.ET_Group.Member1]	:= c_udiSlave1;	(* The Slave1 is the first element of the group c_udiSlaveGroup2 *)
aaudiSubModuleGroups[c_udiSlaveGroup2-TPL.Gc_udiGroupOffset,TPL.ET_Group.Member2]	:= c_udiSlave2;	(* The Slave2 is the second element of the group c_udiSlaveGroup2 *)

(* End of system generated code, could be modified for your application *)


(* System generated code, do not change without consulting 'Schneider Electric Automation GmbH' - otherwise you risk instability!!!*)
xInitSubModulesException := FALSE;

(*****************************************************************************************************************************************************)
(* Set IDs of SubModules *)	

TPL.FC_SetSubModuleIds(	i_udiMainModuleId			:= iq_stStandardModuleItf.i_udiModuleId,
						i_pstSubModulesItf			:= ADR(astSubModuleInterface),
						i_udiNumberOfSubModules		:= c_udiNumberOfSubModules,
						q_etDiag					=> etDiag,
						q_etDiagExt					=> etDiagExtTPL);
					
IF etDiag <> GD.ET_Diag.Ok AND NOT xInitSubModulesException THEN
	xInitSubModulesException := TRUE;
	
	stInitSubModulesException.sMsg := PDL.FC_MultiConcat(	i_sString1 := 'SetSubModuleIds - ', 
															i_sString2 := GD.FC_EtDiagToString(i_etDiag := etDiag), 
															i_sString3 := ' - ', 
															i_sString4 := TPL.FC_EtDiagExtToString(i_etDiagExt := etDiagExtTPL));
END_IF	

(*****************************************************************************************************************************************************)
(* Set exception if any exception occurred *)

TPL.FC_SetException(i_xExceptionActive	:= xInitSubModulesException, 
					iq_stException		:= stInitSubModulesException, 
					iq_stExceptionList	:= iq_stExceptionList, 
					iq_stLogDataList	:= iq_stLogDataList);

xInitSuccessful := xInitSuccessful AND NOT xInitSubModulesException;
					
etDiag := GD.ET_Diag.Ok;
(* End of system generated code, do not change without consulting 'Schneider Electric Automation GmbH' - otherwise you risk instability!!!*)
END_ACTION

ACTION InitModule_Action:
(* This step is used for initialisations after being enabled *)

(* System generated code, could be modified for your application *)
xInitSuccessful := TRUE;

Init_Exceptions();
(* End of system generated code, could be modified for your application *)

(* System generated code, do not change without consulting 'Schneider Electric Automation GmbH' - otherwise you risk instability!!!*)
iq_stStandardModuleItf.q_xActive		:= TRUE;
iq_stStandardModuleItf.q_xReady			:= FALSE;
iq_stStandardModuleItf.q_etDiag			:= GD.ET_Diag.Ok;
iq_stStandardModuleItf.q_udiDiagExt		:= ET_DiagExt.Initializing;
iq_stStandardModuleItf.q_sDiagExt		:= FC_EtDiagExtToString(i_etDiagExt := ET_DiagExt.Initializing);
iq_stStandardModuleItf.q_sMsg			:= '';

Init_SubModules();
Init_CmdTables();
Init_Reactions();
UpdateStructs();
(* End of system generated code, do not change without consulting 'Schneider Electric Automation GmbH' - otherwise you risk instability!!!*)

(* System generated code, could be modified for your application *)
Init_Slave1();
Init_Slave2();
(* End of system generated code, could be modified for your application *)

(* Application specific code *)
(* ToDo: Add your application specific code here *)
;
(* End of application specific code *)
END_ACTION

ACTION Input_Action:
(* System generated code, do not change without consulting 'Schneider Electric Automation GmbH' - otherwise you risk instability!!!*)
UpdateStructs();
(* End of system generated code, do not change without consulting 'Schneider Electric Automation GmbH' - otherwise you risk instability!!!*)
END_ACTION

ACTION Logger_Action:
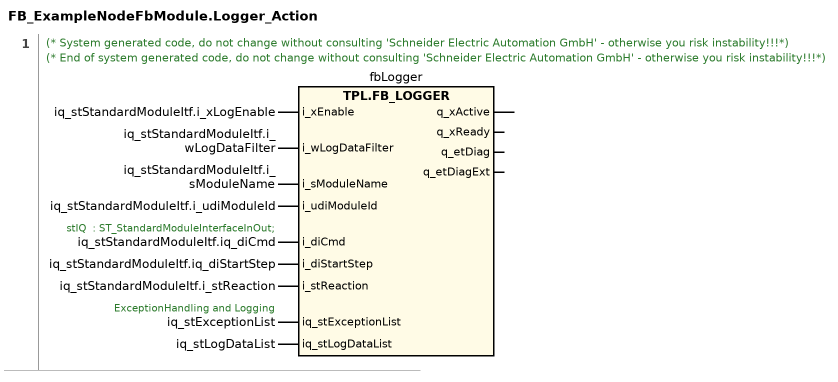
// NETWORK 1
// 					(* System generated code, do not change without consulting 'Schneider Electric Automation GmbH' - otherwise you risk instability!!!*)
// (* End of system generated code, do not change without consulting 'Schneider Electric Automation GmbH' - otherwise you risk instability!!!*)
//
//   fbLogger: Logging related variables
//   iq_stStandardModuleItf.iq_diCmd: stIQ : ST_StandardModuleInterfaceInOut;
//   iq_stExceptionList: ExceptionHandling and Logging
fbLogger(
    i_xEnable := iq_stStandardModuleItf.i_xLogEnable,
    i_wLogDataFilter := iq_stStandardModuleItf.i_wLogDataFilter,
    i_sModuleName := iq_stStandardModuleItf.i_sModuleName,
    i_udiModuleId := iq_stStandardModuleItf.i_udiModuleId,
    i_diCmd := iq_stStandardModuleItf.iq_diCmd,
    i_diStartStep := iq_stStandardModuleItf.iq_diStartStep,
    i_stReaction := iq_stStandardModuleItf.i_stReaction,
    iq_stExceptionList := iq_stExceptionList,
    iq_stLogDataList := iq_stLogDataList); // TPL.FB_LOGGER
END_ACTION

ACTION ModuleFaults:
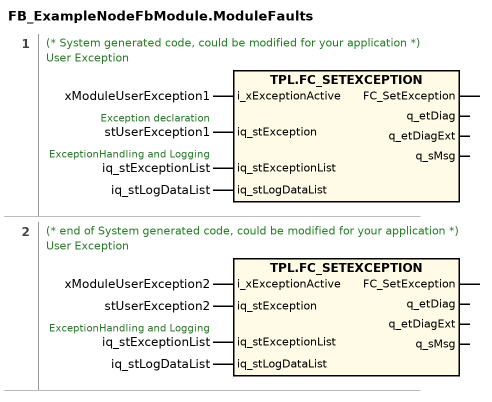
// NETWORK 1
// (* System generated code, could be modified for your application *)
// User Exception
//   stUserException1: Exception declaration
//   iq_stExceptionList: ExceptionHandling and Logging
TPL.FC_SETEXCEPTION(i_xExceptionActive := xModuleUserException1, iq_stException := stUserException1, iq_stExceptionList := iq_stExceptionList, iq_stLogDataList := iq_stLogDataList);

// NETWORK 2
// (* end of System generated code, could be modified for your application *)
// User Exception
//   iq_stExceptionList: ExceptionHandling and Logging
TPL.FC_SETEXCEPTION(i_xExceptionActive := xModuleUserException2, iq_stException := stUserException2, iq_stExceptionList := iq_stExceptionList, iq_stLogDataList := iq_stLogDataList);
END_ACTION

ACTION Output_Active:
(* System generated code, only to be changed by experienced programmers *)
IF iq_stStandardModuleItf.q_udiSubModuleInException <> 0 THEN
	iq_stStandardModuleItf.q_etDiag		:= GD.ET_Diag.Ok;
	iq_stStandardModuleItf.q_udiDiagExt	:= ET_DiagExt.SubModuleInException;
	iq_stStandardModuleItf.q_sDiagExt	:= FC_EtDiagExtToString(i_etDiagExt := ET_DiagExt.SubModuleInException);
	iq_stStandardModuleItf.q_sMsg		:= '';
ELSE
	IF etDiagModuleController = GD.ET_Diag.Ok THEN
		iq_stStandardModuleItf.q_etDiag	:= etDiagModuleController;
		iq_stStandardModuleItf.q_sMsg		:= sMsgModuleController;
		
		CASE etDiagExtModuleController OF
			TPL.ET_DiagExt.DeactivatingSubModules : 
				iq_stStandardModuleItf.q_udiDiagExt	:= ET_DiagExt.DeactivatingSubModules;
				iq_stStandardModuleItf.q_sDiagExt		:= FC_EtDiagExtToString(i_etDiagExt := ET_DiagExt.DeactivatingSubModules);
			TPL.ET_DiagExt.Disabled : 
				iq_stStandardModuleItf.q_udiDiagExt	:= ET_DiagExt.Disabled;
				iq_stStandardModuleItf.q_sDiagExt		:= FC_EtDiagExtToString(i_etDiagExt := ET_DiagExt.Disabled);
			TPL.ET_DiagExt.ExecuteStep : 
				iq_stStandardModuleItf.q_udiDiagExt	:= ET_DiagExt.ExecuteStep;
				iq_stStandardModuleItf.q_sDiagExt		:= FC_EtDiagExtToString(i_etDiagExt := ET_DiagExt.ExecuteStep);
			TPL.ET_DiagExt.Initializing : 
				iq_stStandardModuleItf.q_udiDiagExt	:= ET_DiagExt.Initializing;
				iq_stStandardModuleItf.q_sDiagExt		:= FC_EtDiagExtToString(i_etDiagExt := ET_DiagExt.Initializing);
			TPL.ET_DiagExt.WaitAtNegativeStep : 
				iq_stStandardModuleItf.q_udiDiagExt	:= ET_DiagExt.WaitAtNegativeStep;
				iq_stStandardModuleItf.q_sDiagExt		:= FC_EtDiagExtToString(i_etDiagExt := ET_DiagExt.WaitAtNegativeStep);
			TPL.ET_DiagExt.WaitCmdsDone : 
				iq_stStandardModuleItf.q_udiDiagExt	:= ET_DiagExt.WaitCmdsDone;
				iq_stStandardModuleItf.q_sDiagExt		:= FC_EtDiagExtToString(i_etDiagExt := ET_DiagExt.WaitCmdsDone);
			TPL.ET_DiagExt.WaitForCmd : 
				iq_stStandardModuleItf.q_udiDiagExt	:= ET_DiagExt.WaitForCmd;
				iq_stStandardModuleItf.q_sDiagExt		:= FC_EtDiagExtToString(i_etDiagExt := ET_DiagExt.WaitForCmd);
			ELSE
				iq_stStandardModuleItf.q_etDiag		:= GD. ET_Diag.UnexpectedProgramBehavior;
				iq_stStandardModuleItf.q_udiDiagExt	:= ET_DiagExt.UnknownStateModuleController;
				iq_stStandardModuleItf.q_sDiagExt		:= FC_EtDiagExtToString(i_etDiagExt := ET_DiagExt.UnknownStateModuleController);
		END_CASE
	ELSE
		iq_stStandardModuleItf.q_etDiag		:= GD.ET_Diag.DiagActive;
		iq_stStandardModuleItf.q_udiDiagExt	:= ET_DiagExt.ModuleControllerException;
		iq_stStandardModuleItf.q_sDiagExt	:= FC_EtDiagExtToString(i_etDiagExt := ET_DiagExt.ModuleControllerException);
		iq_stStandardModuleItf.q_sMsg		:= PDL.FC_MultiConcat(	i_sString1 := GD.FC_EtDiagToString(i_etDiag := etDiagModuleController), 
																	i_sString2 := ' - ',
																	i_sString3 := TPL.FC_EtDiagExtToString(i_etDiagExt := etDiagExtModuleController), 
																	i_sString4 := '');
	END_IF
END_IF

(* End of system generated code, only to be changed by experienced programmers *)
END_ACTION

ACTION Start_Action:
(* This step is active until the machine is being enabled *)

(* System generated code, do not change without consulting 'Schneider Electric Automation GmbH' - otherwise you risk instability!!! *)
iq_stStandardModuleItf.q_xActive			:= FALSE;
iq_stStandardModuleItf.q_xReady				:= FALSE;

iq_stStandardModuleItf.q_etDiag				:= GD.ET_Diag.Ok;
iq_stStandardModuleItf.q_udiDiagExt			:= ET_DiagExt.Disabled;
iq_stStandardModuleItf.q_sDiagExt			:= FC_EtDiagExtToString(i_etDiagExt := iq_stStandardModuleItf.q_udiDiagExt);
iq_stStandardModuleItf.q_sMsg				:= '';

iq_stStandardModuleItf.q_dwModuleType		:= TPL.ET_ModuleType.NodeModule;
iq_stStandardModuleItf.q_sModuleTypeName	:= 'NodeModule';
iq_stStandardModuleItf.q_udiModuleVersion	:= 1;	
(* End of system generated code, do not change without consulting 'Schneider Electric Automation GmbH' - otherwise you risk instability!!! *)

(* System generated code, to be changed by experienced programmers *)
IF iq_stStandardModuleItf.iq_diCmd <> 0  AND NOT iq_stStandardModuleItf.i_xEnable THEN
	iq_stStandardModuleItf.iq_diCmd := 0;
END_IF
(* End of system generated code, to be changed by experienced programmers *)

(* Application specific code *)
(* ToDo: Add your application specific code here *)
;
(* End of application specific code *)
END_ACTION

